KUKA KRL program: EPS_2_25716_MHLP06_A_20250905053030.src

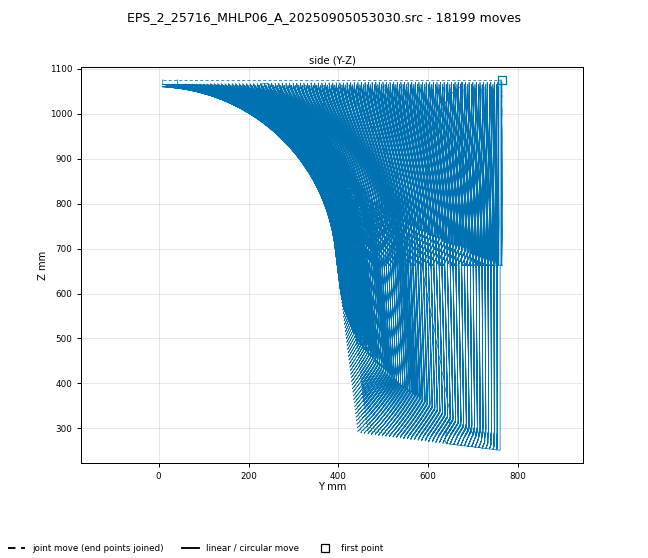
[picture p0: tool path of EPS_2_25716_MHLP06_A_20250905053030.src, 18199 of 18201 moves have a stored position in this frame; points joined in program order, loops and branches not executed]
&ACCESS RVP
&REL 4
&COMMENT QRS 19112012
&PARAM EDITMASK = *
DEF PART()
EXT BAS (BAS_COMMAND :IN,REAL :IN )
INT I
BAS (#INITMOV,0 )

;KUKA QRS Post kuka4.cps  Date:22-06-2017 !

File_ID=2814

QRS_PRE_INIT()

;Init var - Until changes are made in qrs_pre_init
Outlet_Square_prg=0
Inlet_1_Square_prg=0
Inlet_2_Square_prg=0
Inlet_3_Square_prg=0
Inlet_4_Square_prg=0
Inlet_5_Square_prg=0

Outlet_1={X 0.000, Y 514.000, Z 684.500, B 0.000, E1 0.000 }
Inlet_1={X 0.000, Y 514.000, Z 674.500, B 0.000, E1 183.000 }
Outlet_1_type=762
Inlet_1_type=762
;QRS#1=Sidecore dimensions
;QRS#2=750-30" Concrete
;QRS#3=750-30" Concrete
;QRS#4=
;QRS#5=
;QRS#6=
;QRS#7=
;QRS#8=
;QRS#9=S306-42L
;QRS#10=S306-42L
;QRS#11=
;QRS#12=
;QRS#13=
;QRS#14=
;QRS#15=
;QRS#16=1524x152x1524 5'
;QRS#17=EPS Height
;QRS#18=1065,5
;QRS#19=*
;QRS#20= UPDATED VERSION 22-06-2017
;QRS#21=*
Outlet_Square=0550
Inlet_1_Square=0550
Inlet_2_Square=0
Inlet_3_Square=0
Inlet_4_Square=0
Inlet_5_Square=0
Mill_Square=1
Outlet_Square_Prg=266
Inlet_1_Square_prg=266

QRS_INIT()

$ADVANCE=5

; T1
PTP {E1 176.657,E2 176.657}
PTP {X 0,Y 763.394,A -85,B 0,C 180,E1 176.657,E2 176.657,E3 0,E4 0,E5 0,E6 0}
QRS_SPEED_INIT()
LIN {X 0,Y 763.394,Z 1075.5,A -85,B 0,C 180,E1 176.657,E2 176.657,E3 0,E4 0,E5 0,E6 0} C_VEL
LIN {X 0,Y 763.394,Z 665.19,A -85,B 0,C 180,E1 176.657,E2 176.657} C_VEL
LIN {X 0,Y 763.503,Z 663.19,A -85,B 0,C 180,E1 176.807,E2 176.807} C_VEL
LIN {X 0,Y 763.802,Z 663.19,A -85,B 0,C 180,E1 177.187,E2 177.187} C_VEL
LIN {X 0,Y 763.843,Z 663.19,A -85,B 0,C 180,E1 184.692,E2 184.692} C_VEL
LIN {X 0,Y 763.839,Z 663.19,A -85,B 0,C 180,E1 192.28,E2 192.28} C_VEL
LIN {X 0,Y 763.794,Z 663.19,A -85,B 0,C 180,E1 200.096,E2 200.096} C_VEL
LIN {X 0,Y 763.778,Z 663.19,A -85,B 0,C 180,E1 208.327,E2 208.327} C_VEL
LIN {X 0,Y 762.889,Z 663.19,A -85,B 0,C 180,E1 213.338,E2 213.338} C_VEL
LIN {X 0,Y 763.785,Z 663.19,A -85,B 0,C 180,E1 214.937,E2 214.937} C_VEL
LIN {X 0,Y 762.534,Z 663.19,A -85,B 0,C 180,E1 217.329,E2 217.329} C_VEL
LIN {X 0,Y 763.704,Z 663.19,A -85,B 0,C 180,E1 222.138,E2 222.138} C_VEL
LIN {X 0,Y 763.543,Z 663.19,A -85,B 0,C 180,E1 222.564,E2 222.564} C_VEL
LIN {X 0,Y 763.776,Z 663.19,A -85,B 0,C 180,E1 230.266,E2 230.266} C_VEL
LIN {X 0,Y 763.81,Z 663.19,A -85,B 0,C 180,E1 236.912,E2 236.912} C_VEL
LIN {X 0,Y 763.611,Z 663.19,A -85,B 0,C 180,E1 237.107,E2 237.107} C_VEL
LIN {X 0,Y 763.119,Z 663.19,A -85,B 0,C 180,E1 237.178,E2 237.178} C_VEL
LIN {X 0,Y 763.363,Z 714.143,A -85,B 0,C 180,E1 237.755,E2 237.755} C_VEL
LIN {X 0,Y 763.318,Z 729.71,A -85,B 0,C 180,E1 237.961,E2 237.961} C_VEL
LIN {X 0,Y 763.689,Z 748.835,A -85,B 0,C 180,E1 238.314,E2 238.314} C_VEL
LIN {X 0,Y 763.731,Z 766.662,A -85,B 0,C 180,E1 238.702,E2 238.702} C_VEL
LIN {X 0,Y 763.562,Z 784.529,A -85,B 0,C 180,E1 239.155,E2 239.155} C_VEL
LIN {X 0,Y 763.44,Z 791.39,A -85,B 0,C 180,E1 239.353,E2 239.353} C_VEL
LIN {X 0,Y 763.675,Z 803.719,A -85,B 0,C 180,E1 239.742,E2 239.742} C_VEL
LIN {X 0,Y 763.697,Z 820.778,A -85,B 0,C 180,E1 240.333,E2 240.333} C_VEL
LIN {X 0,Y 763.708,Z 837.223,A -85,B 0,C 180,E1 240.974,E2 240.974} C_VEL
LIN {X 0,Y 763.533,Z 854.722,A -85,B 0,C 180,E1 241.73,E2 241.73} C_VEL
LIN {X 0,Y 763.603,Z 871.159,A -85,B 0,C 180,E1 242.528,E2 242.528} C_VEL
LIN {X 0,Y 763.499,Z 886.059,A -85,B 0,C 180,E1 243.314,E2 243.314} C_VEL
LIN {X 0,Y 763.597,Z 901.587,A -85,B 0,C 180,E1 244.22,E2 244.22} C_VEL
LIN {X 0,Y 763.668,Z 915.737,A -85,B 0,C 180,E1 245.118,E2 245.118} C_VEL
LIN {X 0,Y 763.474,Z 930.101,A -85,B 0,C 180,E1 246.101,E2 246.101} C_VEL
LIN {X 0,Y 763.247,Z 942.154,A -85,B 0,C 180,E1 246.988,E2 246.988} C_VEL
LIN {X 0,Y 763.336,Z 956.125,A -85,B 0,C 180,E1 248.123,E2 248.123} C_VEL
LIN {X 0,Y 763.672,Z 967.425,A -85,B 0,C 180,E1 249.12,E2 249.12} C_VEL
LIN {X 0,Y 763.718,Z 974.344,A -85,B 0,C 180,E1 249.772,E2 249.772} C_VEL
LIN {X 0,Y 763.495,Z 980.364,A -85,B 0,C 180,E1 250.349,E2 250.349} C_VEL
LIN {X 0,Y 763.109,Z 990.023,A -85,B 0,C 180,E1 251.332,E2 251.332} C_VEL
LIN {X 0,Y 763.102,Z 1001.366,A -85,B 0,C 180,E1 252.61,E2 252.61} C_VEL
LIN {X 0,Y 763.584,Z 1011.288,A -85,B 0,C 180,E1 253.846,E2 253.846} C_VEL
LIN {X 0,Y 763.803,Z 1015.168,A -85,B 0,C 180,E1 254.372,E2 254.372} C_VEL
LIN {X 0,Y 763.479,Z 1020.327,A -85,B 0,C 180,E1 255.068,E2 255.068} C_VEL
LIN {X 0,Y 762.821,Z 1029.368,A -85,B 0,C 180,E1 256.42,E2 256.42} C_VEL
LIN {X 0,Y 762.79,Z 1036.991,A -85,B 0,C 180,E1 257.703,E2 257.703} C_VEL
LIN {X 0,Y 763.317,Z 1043.373,A -85,B 0,C 180,E1 258.909,E2 258.909} C_VEL
LIN {X 0,Y 763.857,Z 1047.833,A -85,B 0,C 180,E1 259.87,E2 259.87} C_VEL
LIN {X 0,Y 763.425,Z 1050.969,A -85,B 0,C 180,E1 260.578,E2 260.578} C_VEL
LIN {X 0,Y 762.895,Z 1054.781,A -85,B 0,C 180,E1 261.522,E2 261.522} C_VEL
LIN {X 0,Y 762.702,Z 1059.648,A -85,B 0,C 180,E1 262.941,E2 262.941} C_VEL
LIN {X 0,Y 763.282,Z 1063.577,A -85,B 0,C 180,E1 264.362,E2 264.362} C_VEL
LIN {X 0,Y 763.859,Z 1065.587,A -85,B 0,C 180,E1 265.308,E2 265.308} C_VEL
LIN {X 0,Y 763.248,Z 1067.349,A -85,B 0,C 180,E1 266.245,E2 266.245} C_VEL
LIN {X 0,Y 762.721,Z 1068.773,A -85,B 0,C 180,E1 267.183,E2 267.183} C_VEL
LIN {X 0,Y 762.577,Z 1069.998,A -85,B 0,C 180,E1 268.516,E2 268.516} C_VEL
LIN {X 0,Y 762.768,Z 1070.218,A -85,B 0,C 180,E1 269.061,E2 269.061} C_VEL
LIN {X 0,Y 763.872,Z 1070.168,A -85,B 0,C 180,E1 270.937,E2 270.937} C_VEL
LIN {X 0,Y 762.833,Z 1068.771,A -85,B 0,C 180,E1 272.817,E2 272.817} C_VEL
LIN {X 0,Y 762.711,Z 1067.364,A -85,B 0,C 180,E1 273.758,E2 273.758} C_VEL
LIN {X 0,Y 763.16,Z 1064.621,A -85,B 0,C 180,E1 275.167,E2 275.167} C_VEL
LIN {X 0,Y 763.421,Z 1063.574,A -85,B 0,C 180,E1 275.637,E2 275.637} C_VEL
LIN {X 0,Y 763.736,Z 1062.272,A -85,B 0,C 180,E1 276.106,E2 276.106} C_VEL
LIN {X 0,Y 763.75,Z 1060.982,A -85,B 0,C 180,E1 276.577,E2 276.577} C_VEL
LIN {X 0,Y 763.44,Z 1059.643,A -85,B 0,C 180,E1 277.052,E2 277.052} C_VEL
LIN {X 0,Y 762.747,Z 1054.781,A -85,B 0,C 180,E1 278.48,E2 278.48} C_VEL
LIN {X 0,Y 762.808,Z 1048.947,A -85,B 0,C 180,E1 279.905,E2 279.905} C_VEL
LIN {X 0,Y 763.408,Z 1043.373,A -85,B 0,C 180,E1 281.09,E2 281.09} C_VEL
LIN {X 0,Y 763.848,Z 1039.547,A -85,B 0,C 180,E1 281.801,E2 281.801} C_VEL
LIN {X 0,Y 763.464,Z 1035.559,A -85,B 0,C 180,E1 282.541,E2 282.541} C_VEL
LIN {X 0,Y 762.835,Z 1027.394,A -85,B 0,C 180,E1 283.893,E2 283.893} C_VEL
LIN {X 0,Y 762.833,Z 1019.123,A -85,B 0,C 180,E1 285.118,E2 285.118} C_VEL
LIN {X 0,Y 763.436,Z 1009.403,A -85,B 0,C 180,E1 286.402,E2 286.402} C_VEL
LIN {X 0,Y 763.773,Z 1002.371,A -85,B 0,C 180,E1 287.251,E2 287.251} C_VEL
LIN {X 0,Y 763.509,Z 997.07,A -85,B 0,C 180,E1 287.872,E2 287.872} C_VEL
LIN {X 0,Y 763.096,Z 987.878,A -85,B 0,C 180,E1 288.893,E2 288.893} C_VEL
LIN {X 0,Y 762.987,Z 977.021,A -85,B 0,C 180,E1 289.997,E2 289.997} C_VEL
LIN {X 0,Y 763.373,Z 965.026,A -85,B 0,C 180,E1 291.104,E2 291.104} C_VEL
LIN {X 0,Y 763.731,Z 953.245,A -85,B 0,C 180,E1 292.108,E2 292.108} C_VEL
LIN {X 0,Y 763.51,Z 940.467,A -85,B 0,C 180,E1 293.131,E2 293.131} C_VEL
LIN {X 0,Y 763.337,Z 926.48,A -85,B 0,C 180,E1 294.16,E2 294.16} C_VEL
LIN {X 0,Y 763.448,Z 913.778,A -85,B 0,C 180,E1 295.02,E2 295.02} C_VEL
LIN {X 0,Y 763.641,Z 897.91,A -85,B 0,C 180,E1 295.998,E2 295.998} C_VEL
LIN {X 0,Y 763.658,Z 882.443,A -85,B 0,C 180,E1 296.877,E2 296.877} C_VEL
LIN {X 0,Y 763.545,Z 867.236,A -85,B 0,C 180,E1 297.672,E2 297.672} C_VEL
LIN {X 0,Y 763.556,Z 851.419,A -85,B 0,C 180,E1 298.422,E2 298.422} C_VEL
LIN {X 0,Y 763.605,Z 833.293,A -85,B 0,C 180,E1 299.189,E2 299.189} C_VEL
LIN {X 0,Y 763.476,Z 824.344,A -85,B 0,C 180,E1 299.538,E2 299.538} C_VEL
LIN {X 0,Y 763.667,Z 815.688,A -85,B 0,C 180,E1 299.851,E2 299.851} C_VEL
LIN {X 0,Y 763.746,Z 798.997,A -85,B 0,C 180,E1 300.407,E2 300.407} C_VEL
LIN {X 0,Y 763.741,Z 783.59,A -85,B 0,C 180,E1 300.865,E2 300.865} C_VEL
LIN {X 0,Y 763.589,Z 765.456,A -85,B 0,C 180,E1 301.335,E2 301.335} C_VEL
LIN {X 0,Y 763.354,Z 758.258,A -85,B 0,C 180,E1 301.501,E2 301.501} C_VEL
LIN {X 0,Y 763.664,Z 747.28,A -85,B 0,C 180,E1 301.72,E2 301.72} C_VEL
LIN {X 0,Y 763.798,Z 726.383,A -85,B 0,C 180,E1 302.066,E2 302.066} C_VEL
LIN {X 0,Y 763.735,Z 707.916,A -85,B 0,C 180,E1 302.303,E2 302.303} C_VEL
LIN {X 0,Y 763.144,Z 663.19,A -85,B 0,C 180,E1 302.825,E2 302.825} C_VEL
LIN {X 0,Y 763.558,Z 663.19,A -85,B 0,C 180,E1 302.883,E2 302.883} C_VEL
LIN {X 0,Y 763.85,Z 663.19,A -85,B 0,C 180,E1 303.062,E2 303.062} C_VEL
LIN {X 0,Y 763.52,Z 663.19,A -85,B 0,C 180,E1 304.95,E2 304.95} C_VEL
LIN {X 0,Y 763.712,Z 663.19,A -85,B 0,C 180,E1 306.696,E2 306.696} C_VEL
LIN {X 0,Y 763.759,Z 663.19,A -85,B 0,C 180,E1 314.716,E2 314.716} C_VEL
LIN {X 0,Y 763.488,Z 663.19,A -85,B 0,C 180,E1 315.264,E2 315.264} C_VEL
LIN {X 0,Y 763.667,Z 663.19,A -85,B 0,C 180,E1 323.308,E2 323.308} C_VEL
LIN {X 0,Y 762.67,Z 663.19,A -85,B 0,C 180,E1 325.005,E2 325.005} C_VEL
LIN {X 0,Y 762.796,Z 663.19,A -85,B 0,C 180,E1 330.263,E2 330.263} C_VEL
LIN {X 0,Y 763.78,Z 663.19,A -85,B 0,C 180,E1 331.673,E2 331.673} C_VEL
LIN {X 0,Y 763.794,Z 663.19,A -85,B 0,C 180,E1 339.904,E2 339.904} C_VEL
LIN {X 0,Y 763.827,Z 663.19,A -85,B 0,C 180,E1 347.72,E2 347.72} C_VEL
LIN {X 0,Y 763.847,Z 663.19,A -85,B 0,C 180,E1 355.308,E2 355.308} C_VEL
LIN {X 0,Y 763.809,Z 663.19,A -85,B 0,C 180,E1 362.813,E2 362.813} C_VEL
LIN {X 0,Y 763.805,Z 663.19,A -85,B 0,C 180,E1 370.368,E2 370.368} C_VEL
LIN {X 0,Y 763.839,Z 663.19,A -85,B 0,C 180,E1 378.111,E2 378.111} C_VEL
LIN {X 0,Y 762.865,Z 663.19,A -85,B 0,C 180,E1 384.176,E2 384.176} C_VEL
LIN {X 0,Y 763.612,Z 663.19,A -85,B 0,C 180,E1 385.827,E2 385.827} C_VEL
LIN {X 0,Y 763.75,Z 663.19,A -85,B 0,C 180,E1 392.682,E2 392.682} C_VEL
LIN {X 0,Y 763.382,Z 663.19,A -85,B 0,C 180,E1 393.395,E2 393.395} C_VEL
LIN {X 0,Y 763.739,Z 663.19,A -85,B 0,C 180,E1 399.655,E2 399.655} C_VEL
LIN {X 0,Y 763.682,Z 663.19,A -85,B 0,C 180,E1 407.425,E2 407.425} C_VEL
LIN {X 0,Y 763.622,Z 663.19,A -85,B 0,C 180,E1 407.857,E2 407.857} C_VEL
LIN {X 0,Y 763.835,Z 663.19,A -85,B 0,C 180,E1 413.794,E2 413.794} C_VEL
LIN {X 0,Y 763.629,Z 663.19,A -85,B 0,C 180,E1 413.971,E2 413.971} C_VEL
LIN {X 0,Y 761.949,Z 663.19,A -85,B 0,C 180,E1 414.133,E2 414.133} C_VEL
LIN {X 0,Y 762.674,Z 670.746,A -85,B 0,C 180,E1 414.304,E2 414.304} C_VEL
LIN {X 0,Y 763.27,Z 683.05,A -85,B 0,C 180,E1 414.467,E2 414.467} C_VEL
LIN {X 0,Y 763.291,Z 706.143,A -85,B 0,C 180,E1 414.733,E2 414.733} C_VEL
LIN {X 0,Y 763.674,Z 720.884,A -85,B 0,C 180,E1 414.953,E2 414.953} C_VEL
LIN {X 0,Y 763.785,Z 738.788,A -85,B 0,C 180,E1 415.273,E2 415.273} C_VEL
LIN {X 0,Y 763.777,Z 756.953,A -85,B 0,C 180,E1 415.666,E2 415.666} C_VEL
LIN {X 0,Y 763.551,Z 774.753,A -85,B 0,C 180,E1 416.116,E2 416.116} C_VEL
LIN {X 0,Y 763.448,Z 780.911,A -85,B 0,C 180,E1 416.294,E2 416.294} C_VEL
LIN {X 0,Y 763.664,Z 793.266,A -85,B 0,C 180,E1 416.681,E2 416.681} C_VEL
LIN {X 0,Y 763.695,Z 810.232,A -85,B 0,C 180,E1 417.267,E2 417.267} C_VEL
LIN {X 0,Y 763.706,Z 827.815,A -85,B 0,C 180,E1 417.954,E2 417.954} C_VEL
LIN {X 0,Y 763.563,Z 844.112,A -85,B 0,C 180,E1 418.657,E2 418.657} C_VEL
LIN {X 0,Y 763.608,Z 859.823,A -85,B 0,C 180,E1 419.413,E2 419.413} C_VEL
LIN {X 0,Y 763.513,Z 875.27,A -85,B 0,C 180,E1 420.224,E2 420.224} C_VEL
LIN {X 0,Y 763.605,Z 891.803,A -85,B 0,C 180,E1 421.189,E2 421.189} C_VEL
LIN {X 0,Y 763.698,Z 905.659,A -85,B 0,C 180,E1 422.069,E2 422.069} C_VEL
LIN {X 0,Y 763.535,Z 919.141,A -85,B 0,C 180,E1 422.987,E2 422.987} C_VEL
LIN {X 0,Y 763.26,Z 932.57,A -85,B 0,C 180,E1 423.977,E2 423.977} C_VEL
LIN {X 0,Y 763.327,Z 945.733,A -85,B 0,C 180,E1 425.044,E2 425.044} C_VEL
LIN {X 0,Y 763.668,Z 957.774,A -85,B 0,C 180,E1 426.108,E2 426.108} C_VEL
LIN {X 0,Y 763.749,Z 964.577,A -85,B 0,C 180,E1 426.75,E2 426.75} C_VEL
LIN {X 0,Y 763.488,Z 971.081,A -85,B 0,C 180,E1 427.378,E2 427.378} C_VEL
LIN {X 0,Y 763.087,Z 979.912,A -85,B 0,C 180,E1 428.274,E2 428.274} C_VEL
LIN {X 0,Y 762.976,Z 990.113,A -85,B 0,C 180,E1 429.41,E2 429.41} C_VEL
LIN {X 0,Y 763.479,Z 1001.309,A -85,B 0,C 180,E1 430.801,E2 430.801} C_VEL
LIN {X 0,Y 763.844,Z 1007.354,A -85,B 0,C 180,E1 431.62,E2 431.62} C_VEL
LIN {X 0,Y 763.573,Z 1011.028,A -85,B 0,C 180,E1 432.129,E2 432.129} C_VEL
LIN {X 0,Y 762.949,Z 1019.161,A -85,B 0,C 180,E1 433.343,E2 433.343} C_VEL
LIN {X 0,Y 762.76,Z 1025.695,A -85,B 0,C 180,E1 434.425,E2 434.425} C_VEL
LIN {X 0,Y 763.186,Z 1032.951,A -85,B 0,C 180,E1 435.781,E2 435.781} C_VEL
LIN {X 0,Y 763.744,Z 1037.559,A -85,B 0,C 180,E1 436.765,E2 436.765} C_VEL
LIN {X 0,Y 763.737,Z 1039.417,A -85,B 0,C 180,E1 437.162,E2 437.162} C_VEL
LIN {X 0,Y 762.866,Z 1045.491,A -85,B 0,C 180,E1 438.663,E2 438.663} C_VEL
LIN {X 0,Y 762.68,Z 1050.25,A -85,B 0,C 180,E1 440.093,E2 440.093} C_VEL
LIN {X 0,Y 763.274,Z 1054.066,A -85,B 0,C 180,E1 441.526,E2 441.526} C_VEL
LIN {X 0,Y 763.845,Z 1056.046,A -85,B 0,C 180,E1 442.479,E2 442.479} C_VEL
LIN {X 0,Y 763.25,Z 1057.677,A -85,B 0,C 180,E1 443.419,E2 443.419} C_VEL
LIN {X 0,Y 762.729,Z 1059.001,A -85,B 0,C 180,E1 444.358,E2 444.358} C_VEL
LIN {X 0,Y 762.57,Z 1059.845,A -85,B 0,C 180,E1 445.3,E2 445.3} C_VEL
LIN {X 0,Y 762.768,Z 1060.283,A -85,B 0,C 180,E1 446.236,E2 446.236} C_VEL
LIN {X 0,Y 763.261,Z 1060.412,A -85,B 0,C 180,E1 447.185,E2 447.185} C_VEL
LIN {X 0,Y 763.773,Z 1060.049,A -85,B 0,C 180,E1 448.312,E2 448.312} C_VEL
LIN {X 0,Y 762.916,Z 1058.708,A -85,B 0,C 180,E1 449.812,E2 449.812} C_VEL
LIN {X 0,Y 762.704,Z 1057.026,A -85,B 0,C 180,E1 450.939,E2 450.939} C_VEL
LIN {X 0,Y 763.033,Z 1054.747,A -85,B 0,C 180,E1 452.065,E2 452.065} C_VEL
LIN {X 0,Y 763.434,Z 1052.961,A -85,B 0,C 180,E1 452.815,E2 452.815} C_VEL
LIN {X 0,Y 763.825,Z 1050.803,A -85,B 0,C 180,E1 453.596,E2 453.596} C_VEL
LIN {X 0,Y 763.187,Z 1047.332,A -85,B 0,C 180,E1 454.696,E2 454.696} C_VEL
LIN {X 0,Y 762.935,Z 1045.751,A -85,B 0,C 180,E1 455.169,E2 455.169} C_VEL
LIN {X 0,Y 762.766,Z 1039.129,A -85,B 0,C 180,E1 456.822,E2 456.822} C_VEL
LIN {X 0,Y 763.285,Z 1033.601,A -85,B 0,C 180,E1 458,E2 458} C_VEL
LIN {X 0,Y 763.86,Z 1028.555,A -85,B 0,C 180,E1 458.941,E2 458.941} C_VEL
LIN {X 0,Y 763.483,Z 1024.574,A -85,B 0,C 180,E1 459.659,E2 459.659} C_VEL
LIN {X 0,Y 762.931,Z 1017.317,A -85,B 0,C 180,E1 460.858,E2 460.858} C_VEL
LIN {X 0,Y 762.854,Z 1009.247,A -85,B 0,C 180,E1 462.056,E2 462.056} C_VEL
LIN {X 0,Y 763.43,Z 998.964,A -85,B 0,C 180,E1 463.41,E2 463.41} C_VEL
LIN {X 0,Y 763.814,Z 992.361,A -85,B 0,C 180,E1 464.207,E2 464.207} C_VEL
LIN {X 0,Y 763.552,Z 986.364,A -85,B 0,C 180,E1 464.905,E2 464.905} C_VEL
LIN {X 0,Y 763.202,Z 978.727,A -85,B 0,C 180,E1 465.759,E2 465.759} C_VEL
LIN {X 0,Y 763.026,Z 967.557,A -85,B 0,C 180,E1 466.901,E2 466.901} C_VEL
LIN {X 0,Y 763.363,Z 955.721,A -85,B 0,C 180,E1 467.999,E2 467.999} C_VEL
LIN {X 0,Y 763.745,Z 942.465,A -85,B 0,C 180,E1 469.125,E2 469.125} C_VEL
LIN {X 0,Y 763.517,Z 930.218,A -85,B 0,C 180,E1 470.104,E2 470.104} C_VEL
LIN {X 0,Y 763.287,Z 916.729,A -85,B 0,C 180,E1 471.1,E2 471.1} C_VEL
LIN {X 0,Y 763.377,Z 902.542,A -85,B 0,C 180,E1 472.055,E2 472.055} C_VEL
LIN {X 0,Y 763.626,Z 888.226,A -85,B 0,C 180,E1 472.936,E2 472.936} C_VEL
LIN {X 0,Y 763.684,Z 872.5,A -85,B 0,C 180,E1 473.828,E2 473.828} C_VEL
LIN {X 0,Y 763.623,Z 856.934,A -85,B 0,C 180,E1 474.639,E2 474.639} C_VEL
LIN {X 0,Y 763.629,Z 840.802,A -85,B 0,C 180,E1 475.4,E2 475.4} C_VEL
LIN {X 0,Y 763.624,Z 823.946,A -85,B 0,C 180,E1 476.118,E2 476.118} C_VEL
LIN {X 0,Y 763.519,Z 814.426,A -85,B 0,C 180,E1 476.489,E2 476.489} C_VEL
LIN {X 0,Y 763.706,Z 805.542,A -85,B 0,C 180,E1 476.809,E2 476.809} C_VEL
LIN {X 0,Y 763.748,Z 788.836,A -85,B 0,C 180,E1 477.367,E2 477.367} C_VEL
LIN {X 0,Y 763.74,Z 771.331,A -85,B 0,C 180,E1 477.88,E2 477.88} C_VEL
LIN {X 0,Y 763.608,Z 752.724,A -85,B 0,C 180,E1 478.35,E2 478.35} C_VEL
LIN {X 0,Y 763.364,Z 742.185,A -85,B 0,C 180,E1 478.585,E2 478.585} C_VEL
LIN {X 0,Y 763.599,Z 733.423,A -85,B 0,C 180,E1 478.746,E2 478.746} C_VEL
LIN {X 0,Y 763.746,Z 718.002,A -85,B 0,C 180,E1 479.002,E2 479.002} C_VEL
LIN {X 0,Y 763.66,Z 695.951,A -85,B 0,C 180,E1 479.283,E2 479.283} C_VEL
LIN {X 0,Y 763.248,Z 663.19,A -85,B 0,C 180,E1 479.663,E2 479.663} C_VEL
LIN {X 0,Y 763.483,Z 663.19,A -85,B 0,C 180,E1 479.696,E2 479.696} C_VEL
LIN {X 0,Y 763.798,Z 663.19,A -85,B 0,C 180,E1 479.868,E2 479.868} C_VEL
LIN {X 0,Y 762.898,Z 663.19,A -85,B 0,C 180,E1 484.983,E2 484.983} C_VEL
LIN {X 0,Y 763.644,Z 663.19,A -85,B 0,C 180,E1 486.689,E2 486.689} C_VEL
LIN {X 0,Y 763.687,Z 663.19,A -85,B 0,C 180,E1 494.721,E2 494.721} C_VEL
LIN {X 0,Y 763.478,Z 663.19,A -85,B 0,C 180,E1 495.263,E2 495.263} C_VEL
LIN {X 0,Y 762.367,Z 663.19,A -85,B 0,C 180,E1 500.394,E2 500.394} C_VEL
LIN {X 0,Y 763.72,Z 663.19,A -85,B 0,C 180,E1 502.739,E2 502.739} C_VEL
LIN {X 0,Y 763.638,Z 663.19,A -85,B 0,C 180,E1 510.152,E2 510.152} C_VEL
LIN {X 0,Y 762.933,Z 663.19,A -85,B 0,C 180,E1 511.639,E2 511.639} C_VEL
LIN {X 0,Y 763.821,Z 663.19,A -85,B 0,C 180,E1 517.895,E2 517.895} C_VEL
LIN {X 0,Y 763.451,Z 663.19,A -85,B 0,C 180,E1 524.967,E2 524.967} C_VEL
LIN {X 0,Y 763.654,Z 663.19,A -85,B 0,C 180,E1 525.79,E2 525.79} C_VEL
LIN {X 0,Y 763.811,Z 663.19,A -85,B 0,C 180,E1 529.632,E2 529.632} C_VEL
LIN {X 0,Y 763.503,Z 663.19,A -85,B 0,C 180,E1 536.807,E2 536.807} C_VEL
LIN {X 0,Y 754.48,Z 663.19,A -85,B 0,C 180,E1 539.404,E2 539.404} C_VEL
LIN {X 0,Y 754.687,Z 663.19,A -85,B 0,C 180,E1 546.363,E2 546.363} C_VEL
LIN {X 0,Y 754.972,Z 663.19,A -85,B 0,C 180,E1 553.38,E2 553.38} C_VEL
LIN {X 0,Y 755.058,Z 663.19,A -85,B 0,C 180,E1 560.953,E2 560.953} C_VEL
LIN {X 0,Y 755.058,Z 663.19,A -85,B 0,C 180,E1 569.519,E2 569.519} C_VEL
LIN {X 0,Y 754.873,Z 663.19,A -85,B 0,C 180,E1 576.396,E2 576.396} C_VEL
LIN {X 0,Y 755.272,Z 663.19,A -85,B 0,C 180,E1 582.876,E2 582.876} C_VEL
LIN {X 0,Y 755.409,Z 663.19,A -85,B 0,C 180,E1 590.778,E2 590.778} C_VEL
LIN {X 0,Y 755.916,Z 664.759,A -85,B 0,C 180,E1 596.843,E2 596.843} C_VEL
LIN {X 0,Y 756.868,Z 759.718,A -85,B 0,C 180,E1 598.229,E2 598.229} C_VEL
LIN {X 0,Y 756.569,Z 829.969,A -85,B 0,C 180,E1 600.384,E2 600.384} C_VEL
LIN {X 0,Y 756.114,Z 898.18,A -85,B 0,C 180,E1 603.739,E2 603.739} C_VEL
LIN {X 0,Y 755.607,Z 957.987,A -85,B 0,C 180,E1 608.051,E2 608.051} C_VEL
LIN {X 0,Y 755.379,Z 1006.638,A -85,B 0,C 180,E1 613.077,E2 613.077} C_VEL
LIN {X 0,Y 755.094,Z 1041.42,A -85,B 0,C 180,E1 618.415,E2 618.415} C_VEL
LIN {X 0,Y 754.949,Z 1061.847,A -85,B 0,C 180,E1 623.658,E2 623.658} C_VEL
LIN {X 0,Y 754.595,Z 1069.802,A -85,B 0,C 180,E1 628.273,E2 628.273} C_VEL
LIN {X 0,Y 754.847,Z 1068.731,A -85,B 0,C 180,E1 632.879,E2 632.879} C_VEL
LIN {X 0,Y 755.199,Z 1058.413,A -85,B 0,C 180,E1 637.5,E2 637.5} C_VEL
LIN {X 0,Y 755.225,Z 1033.216,A -85,B 0,C 180,E1 643.073,E2 643.073} C_VEL
LIN {X 0,Y 755.422,Z 993.868,A -85,B 0,C 180,E1 648.431,E2 648.431} C_VEL
LIN {X 0,Y 755.875,Z 942.929,A -85,B 0,C 180,E1 653.186,E2 653.186} C_VEL
LIN {X 0,Y 756.271,Z 881.314,A -85,B 0,C 180,E1 657.221,E2 657.221} C_VEL
LIN {X 0,Y 756.618,Z 813.428,A -85,B 0,C 180,E1 660.236,E2 660.236} C_VEL
LIN {X 0,Y 756.926,Z 740.759,A -85,B 0,C 180,E1 662.151,E2 662.151} C_VEL
LIN {X 0,Y 755.817,Z 663.19,A -85,B 0,C 180,E1 663.186,E2 663.186} C_VEL
LIN {X 0,Y 754.086,Z 663.19,A -85,B 0,C 180,E1 669.305,E2 669.305} C_VEL
LIN {X 0,Y 754.833,Z 663.19,A -85,B 0,C 180,E1 676.058,E2 676.058} C_VEL
LIN {X 0,Y 754.921,Z 663.19,A -85,B 0,C 180,E1 684.442,E2 684.442} C_VEL
LIN {X 0,Y 755.641,Z 663.19,A -85,B 0,C 180,E1 691.82,E2 691.82} C_VEL
LIN {X 0,Y 755.202,Z 663.19,A -85,B 0,C 180,E1 700.62,E2 700.62} C_VEL
LIN {X 0,Y 754.916,Z 663.19,A -85,B 0,C 180,E1 708.976,E2 708.976} C_VEL
LIN {X 0,Y 755.342,Z 663.19,A -85,B 0,C 180,E1 715.955,E2 715.955} C_VEL
LIN {X 0,Y 754.915,Z 663.19,A -85,B 0,C 180,E1 724.023,E2 724.023} C_VEL
LIN {X 0,Y 755.309,Z 663.19,A -85,B 0,C 180,E1 730.993,E2 730.993} C_VEL
LIN {X 0,Y 754.961,Z 663.19,A -85,B 0,C 180,E1 739.36,E2 739.36} C_VEL
LIN {X 0,Y 754.93,Z 663.19,A -85,B 0,C 180,E1 746.881,E2 746.881} C_VEL
LIN {X 0,Y 755.271,Z 663.19,A -85,B 0,C 180,E1 753.568,E2 753.568} C_VEL
LIN {X 0,Y 754.686,Z 663.19,A -85,B 0,C 180,E1 761.105,E2 761.105} C_VEL
LIN {X 0,Y 755.062,Z 663.19,A -85,B 0,C 180,E1 768.902,E2 768.902} C_VEL
LIN {X 0,Y 754.972,Z 663.19,A -85,B 0,C 180,E1 773.838,E2 773.838} C_VEL
LIN {X 0,Y 756.929,Z 755.494,A -85,B 0,C 180,E1 775.313,E2 775.313} C_VEL
LIN {X 0,Y 756.585,Z 826.044,A -85,B 0,C 180,E1 777.578,E2 777.578} C_VEL
LIN {X 0,Y 756.13,Z 892.372,A -85,B 0,C 180,E1 780.952,E2 780.952} C_VEL
LIN {X 0,Y 755.702,Z 952.369,A -85,B 0,C 180,E1 785.394,E2 785.394} C_VEL
LIN {X 0,Y 755.483,Z 1000.435,A -85,B 0,C 180,E1 790.506,E2 790.506} C_VEL
LIN {X 0,Y 755.342,Z 1034.832,A -85,B 0,C 180,E1 796.059,E2 796.059} C_VEL
LIN {X 0,Y 755.482,Z 1055.025,A -85,B 0,C 180,E1 801.923,E2 801.923} C_VEL
LIN {X 0,Y 755.24,Z 1060.458,A -85,B 0,C 180,E1 807.122,E2 807.122} C_VEL
LIN {X 0,Y 755.477,Z 1052.976,A -85,B 0,C 180,E1 812.876,E2 812.876} C_VEL
LIN {X 0,Y 755.692,Z 1030.759,A -85,B 0,C 180,E1 818.656,E2 818.656} C_VEL
LIN {X 0,Y 755.905,Z 993.718,A -85,B 0,C 180,E1 824.226,E2 824.226} C_VEL
LIN {X 0,Y 756.037,Z 944.765,A -85,B 0,C 180,E1 829.174,E2 829.174} C_VEL
LIN {X 0,Y 756.205,Z 884.806,A -85,B 0,C 180,E1 833.409,E2 833.409} C_VEL
LIN {X 0,Y 756.415,Z 815.296,A -85,B 0,C 180,E1 836.76,E2 836.76} C_VEL
LIN {X 0,Y 756.577,Z 740.886,A -85,B 0,C 180,E1 838.93,E2 838.93} C_VEL
LIN {X 0,Y 755.622,Z 663.19,A -85,B 0,C 180,E1 840.119,E2 840.119} C_VEL
LIN {X 0,Y 754.751,Z 663.19,A -85,B 0,C 180,E1 847.791,E2 847.791} C_VEL
LIN {X 0,Y 754.876,Z 663.19,A -85,B 0,C 180,E1 856.096,E2 856.096} C_VEL
LIN {X 0,Y 755.027,Z 663.19,A -85,B 0,C 180,E1 863.644,E2 863.644} C_VEL
LIN {X 0,Y 754.844,Z 663.19,A -85,B 0,C 180,E1 871.816,E2 871.816} C_VEL
LIN {X 0,Y 754.774,Z 663.19,A -85,B 0,C 180,E1 879.409,E2 879.409} C_VEL
LIN {X 0,Y 755.383,Z 663.19,A -85,B 0,C 180,E1 886.811,E2 886.811} C_VEL
LIN {X 0,Y 754.166,Z 663.19,A -85,B 0,C 180,E1 893.658,E2 893.658} C_VEL
LIN {X 0,Y 755.008,Z 663.19,A -85,B 0,C 180,E1 898.285,E2 898.285} C_VEL
LIN {X 0,Y 754.48,Z 663.19,A -85,B 0,C 180,E1 899.404,E2 899.404} C_VEL
LIN {X 0,Y 746.358,Z 663.19,A -85,B 0,C 180,E1 902.034,E2 902.034} C_VEL
LIN {X 0,Y 746.257,Z 663.19,A -85,B 0,C 180,E1 907.61,E2 907.61} C_VEL
LIN {X 0,Y 746.872,Z 663.19,A -85,B 0,C 180,E1 913.528,E2 913.528} C_VEL
LIN {X 0,Y 747.144,Z 663.19,A -85,B 0,C 180,E1 920.838,E2 920.838} C_VEL
LIN {X 0,Y 747.49,Z 663.19,A -85,B 0,C 180,E1 928.515,E2 928.515} C_VEL
LIN {X 0,Y 747.446,Z 663.19,A -85,B 0,C 180,E1 935.377,E2 935.377} C_VEL
LIN {X 0,Y 747.243,Z 663.19,A -85,B 0,C 180,E1 942.896,E2 942.896} C_VEL
LIN {X 0,Y 746.902,Z 663.19,A -85,B 0,C 180,E1 951.74,E2 951.74} C_VEL
LIN {X 0,Y 747.708,Z 665.181,A -85,B 0,C 180,E1 956.436,E2 956.436} C_VEL
LIN {X 0,Y 749.825,Z 699.861,A -85,B 0,C 180,E1 956.932,E2 956.932} C_VEL
LIN {X 0,Y 749.856,Z 774.935,A -85,B 0,C 180,E1 958.271,E2 958.271} C_VEL
LIN {X 0,Y 749.273,Z 845.914,A -85,B 0,C 180,E1 960.743,E2 960.743} C_VEL
LIN {X 0,Y 748.603,Z 911.358,A -85,B 0,C 180,E1 964.293,E2 964.293} C_VEL
LIN {X 0,Y 748.101,Z 969.045,A -85,B 0,C 180,E1 968.82,E2 968.82} C_VEL
LIN {X 0,Y 747.915,Z 1015.785,A -85,B 0,C 180,E1 974.115,E2 974.115} C_VEL
LIN {X 0,Y 747.661,Z 1047.079,A -85,B 0,C 180,E1 979.483,E2 979.483} C_VEL
LIN {X 0,Y 747.775,Z 1065.919,A -85,B 0,C 180,E1 985.348,E2 985.348} C_VEL
LIN {X 0,Y 747.602,Z 1070.338,A -85,B 0,C 180,E1 990.581,E2 990.581} C_VEL
LIN {X 0,Y 747.718,Z 1061.845,A -85,B 0,C 180,E1 996.405,E2 996.405} C_VEL
LIN {X 0,Y 747.658,Z 1038.316,A -85,B 0,C 180,E1 1002.296,E2 1002.296} C_VEL
LIN {X 0,Y 747.847,Z 1001.03,A -85,B 0,C 180,E1 1007.799,E2 1007.799} C_VEL
LIN {X 0,Y 748.229,Z 950.883,A -85,B 0,C 180,E1 1012.784,E2 1012.784} C_VEL
LIN {X 0,Y 748.843,Z 890.489,A -85,B 0,C 180,E1 1016.99,E2 1016.99} C_VEL
LIN {X 0,Y 749.401,Z 822.492,A -85,B 0,C 180,E1 1020.224,E2 1020.224} C_VEL
LIN {X 0,Y 749.952,Z 749.891,A -85,B 0,C 180,E1 1022.313,E2 1022.313} C_VEL
LIN {X 0,Y 748.098,Z 665.576,A -85,B 0,C 180,E1 1023.54,E2 1023.54} C_VEL
LIN {X 0,Y 747.646,Z 663.19,A -85,B 0,C 180,E1 1023.902,E2 1023.902} C_VEL
LIN {X 0,Y 746.095,Z 663.19,A -85,B 0,C 180,E1 1032.034,E2 1032.034} C_VEL
LIN {X 0,Y 746.774,Z 663.19,A -85,B 0,C 180,E1 1036.127,E2 1036.127} C_VEL
LIN {X 0,Y 746.86,Z 663.19,A -85,B 0,C 180,E1 1044.591,E2 1044.591} C_VEL
LIN {X 0,Y 746.864,Z 663.19,A -85,B 0,C 180,E1 1052.776,E2 1052.776} C_VEL
LIN {X 0,Y 747.163,Z 663.19,A -85,B 0,C 180,E1 1060.691,E2 1060.691} C_VEL
LIN {X 0,Y 746.994,Z 663.19,A -85,B 0,C 180,E1 1068.858,E2 1068.858} C_VEL
LIN {X 0,Y 747.357,Z 663.19,A -85,B 0,C 180,E1 1075.911,E2 1075.911} C_VEL
LIN {X 0,Y 746.882,Z 663.19,A -85,B 0,C 180,E1 1084.066,E2 1084.066} C_VEL
LIN {X 0,Y 747.221,Z 663.19,A -85,B 0,C 180,E1 1091.113,E2 1091.113} C_VEL
LIN {X 0,Y 746.849,Z 663.19,A -85,B 0,C 180,E1 1099.579,E2 1099.579} C_VEL
LIN {X 0,Y 746.772,Z 663.19,A -85,B 0,C 180,E1 1107.199,E2 1107.199} C_VEL
LIN {X 0,Y 746.743,Z 663.19,A -85,B 0,C 180,E1 1114.67,E2 1114.67} C_VEL
LIN {X 0,Y 746.554,Z 663.19,A -85,B 0,C 180,E1 1121.34,E2 1121.34} C_VEL
LIN {X 0,Y 747.129,Z 663.19,A -85,B 0,C 180,E1 1128.727,E2 1128.727} C_VEL
LIN {X 0,Y 747.748,Z 664.557,A -85,B 0,C 180,E1 1133.498,E2 1133.498} C_VEL
LIN {X 0,Y 750.031,Z 757.212,A -85,B 0,C 180,E1 1135.033,E2 1135.033} C_VEL
LIN {X 0,Y 749.44,Z 826.899,A -85,B 0,C 180,E1 1137.308,E2 1137.308} C_VEL
LIN {X 0,Y 748.676,Z 893.608,A -85,B 0,C 180,E1 1140.753,E2 1140.753} C_VEL
LIN {X 0,Y 747.955,Z 953.013,A -85,B 0,C 180,E1 1145.216,E2 1145.216} C_VEL
LIN {X 0,Y 747.532,Z 1000.165,A -85,B 0,C 180,E1 1150.29,E2 1150.29} C_VEL
LIN {X 0,Y 747.315,Z 1034.676,A -85,B 0,C 180,E1 1155.907,E2 1155.907} C_VEL
LIN {X 0,Y 747.453,Z 1054.956,A -85,B 0,C 180,E1 1161.835,E2 1161.835} C_VEL
LIN {X 0,Y 747.215,Z 1060.468,A -85,B 0,C 180,E1 1167.092,E2 1167.092} C_VEL
LIN {X 0,Y 747.505,Z 1053.064,A -85,B 0,C 180,E1 1172.907,E2 1172.907} C_VEL
LIN {X 0,Y 747.757,Z 1030.935,A -85,B 0,C 180,E1 1178.748,E2 1178.748} C_VEL
LIN {X 0,Y 748.004,Z 993.998,A -85,B 0,C 180,E1 1184.379,E2 1184.379} C_VEL
LIN {X 0,Y 748.314,Z 945.84,A -85,B 0,C 180,E1 1189.32,E2 1189.32} C_VEL
LIN {X 0,Y 748.795,Z 886.394,A -85,B 0,C 180,E1 1193.598,E2 1193.598} C_VEL
LIN {X 0,Y 749.292,Z 817.869,A -85,B 0,C 180,E1 1196.971,E2 1196.971} C_VEL
LIN {X 0,Y 749.684,Z 743.698,A -85,B 0,C 180,E1 1199.198,E2 1199.198} C_VEL
LIN {X 0,Y 748.299,Z 666.762,A -85,B 0,C 180,E1 1200.359,E2 1200.359} C_VEL
LIN {X 0,Y 747.354,Z 663.19,A -85,B 0,C 180,E1 1200.536,E2 1200.536} C_VEL
LIN {X 0,Y 746.341,Z 663.19,A -85,B 0,C 180,E1 1208.489,E2 1208.489} C_VEL
LIN {X 0,Y 746.854,Z 663.19,A -85,B 0,C 180,E1 1216.119,E2 1216.119} C_VEL
LIN {X 0,Y 747.147,Z 663.19,A -85,B 0,C 180,E1 1223.292,E2 1223.292} C_VEL
LIN {X 0,Y 746.733,Z 663.19,A -85,B 0,C 180,E1 1232.051,E2 1232.051} C_VEL
LIN {X 0,Y 746.917,Z 663.19,A -85,B 0,C 180,E1 1239.183,E2 1239.183} C_VEL
LIN {X 0,Y 747.334,Z 663.19,A -85,B 0,C 180,E1 1247.7,E2 1247.7} C_VEL
LIN {X 0,Y 747.724,Z 663.19,A -85,B 0,C 180,E1 1257.104,E2 1257.104} C_VEL
LIN {X 0,Y 746.358,Z 663.19,A -85,B 0,C 180,E1 1262.034,E2 1262.034} C_VEL
LIN {X 0,Y 739.292,Z 663.19,A -85,B 0,C 180,E1 1264.716,E2 1264.716} C_VEL
LIN {X 0,Y 738.776,Z 663.19,A -85,B 0,C 180,E1 1273.679,E2 1273.679} C_VEL
LIN {X 0,Y 738.951,Z 663.19,A -85,B 0,C 180,E1 1281.08,E2 1281.08} C_VEL
LIN {X 0,Y 739.107,Z 663.19,A -85,B 0,C 180,E1 1289.313,E2 1289.313} C_VEL
LIN {X 0,Y 739.158,Z 663.19,A -85,B 0,C 180,E1 1295.87,E2 1295.87} C_VEL
LIN {X 0,Y 738.836,Z 663.19,A -85,B 0,C 180,E1 1303.504,E2 1303.504} C_VEL
LIN {X 0,Y 739.061,Z 663.19,A -85,B 0,C 180,E1 1311.259,E2 1311.259} C_VEL
LIN {X 0,Y 739.37,Z 664.769,A -85,B 0,C 180,E1 1316.001,E2 1316.001} C_VEL
LIN {X 0,Y 743.086,Z 678.117,A -85,B 0,C 180,E1 1316.346,E2 1316.346} C_VEL
LIN {X 0,Y 743.192,Z 762.398,A -85,B 0,C 180,E1 1317.632,E2 1317.632} C_VEL
LIN {X 0,Y 742.349,Z 832.082,A -85,B 0,C 180,E1 1319.842,E2 1319.842} C_VEL
LIN {X 0,Y 741.245,Z 900.309,A -85,B 0,C 180,E1 1323.301,E2 1323.301} C_VEL
LIN {X 0,Y 740.163,Z 959.751,A -85,B 0,C 180,E1 1327.727,E2 1327.727} C_VEL
LIN {X 0,Y 739.569,Z 1007.861,A -85,B 0,C 180,E1 1332.858,E2 1332.858} C_VEL
LIN {X 0,Y 739.213,Z 1042.968,A -85,B 0,C 180,E1 1338.463,E2 1338.463} C_VEL
LIN {X 0,Y 739.175,Z 1063.415,A -85,B 0,C 180,E1 1344.113,E2 1344.113} C_VEL
LIN {X 0,Y 738.928,Z 1070.338,A -85,B 0,C 180,E1 1349.412,E2 1349.412} C_VEL
LIN {X 0,Y 739.097,Z 1065.331,A -85,B 0,C 180,E1 1354.995,E2 1354.995} C_VEL
LIN {X 0,Y 739.191,Z 1047.075,A -85,B 0,C 180,E1 1360.64,E2 1360.64} C_VEL
LIN {X 0,Y 739.499,Z 1014.681,A -85,B 0,C 180,E1 1366.224,E2 1366.224} C_VEL
LIN {X 0,Y 740.175,Z 968.384,A -85,B 0,C 180,E1 1371.482,E2 1371.482} C_VEL
LIN {X 0,Y 741.068,Z 910.926,A -85,B 0,C 180,E1 1376.016,E2 1376.016} C_VEL
LIN {X 0,Y 742.052,Z 843.203,A -85,B 0,C 180,E1 1379.691,E2 1379.691} C_VEL
LIN {X 0,Y 742.92,Z 770.56,A -85,B 0,C 180,E1 1382.176,E2 1382.176} C_VEL
LIN {X 0,Y 743.285,Z 689.976,A -85,B 0,C 180,E1 1383.509,E2 1383.509} C_VEL
LIN {X 0,Y 741.024,Z 667.635,A -85,B 0,C 180,E1 1383.88,E2 1383.88} C_VEL
LIN {X 0,Y 739.631,Z 663.19,A -85,B 0,C 180,E1 1384.071,E2 1384.071} C_VEL
LIN {X 0,Y 738.78,Z 663.19,A -85,B 0,C 180,E1 1393.442,E2 1393.442} C_VEL
LIN {X 0,Y 738.884,Z 663.19,A -85,B 0,C 180,E1 1402.685,E2 1402.685} C_VEL
LIN {X 0,Y 739.077,Z 663.19,A -85,B 0,C 180,E1 1412.465,E2 1412.465} C_VEL
LIN {X 0,Y 738.715,Z 663.19,A -85,B 0,C 180,E1 1421.416,E2 1421.416} C_VEL
LIN {X 0,Y 739.042,Z 663.19,A -85,B 0,C 180,E1 1428.736,E2 1428.736} C_VEL
LIN {X 0,Y 739.353,Z 663.19,A -85,B 0,C 180,E1 1435.867,E2 1435.867} C_VEL
LIN {X 0,Y 738.851,Z 663.19,A -85,B 0,C 180,E1 1444.11,E2 1444.11} C_VEL
LIN {X 0,Y 739.122,Z 663.19,A -85,B 0,C 180,E1 1451.237,E2 1451.237} C_VEL
LIN {X 0,Y 739.471,Z 663.19,A -85,B 0,C 180,E1 1458.537,E2 1458.537} C_VEL
LIN {X 0,Y 738.903,Z 663.19,A -85,B 0,C 180,E1 1466.781,E2 1466.781} C_VEL
LIN {X 0,Y 738.856,Z 663.19,A -85,B 0,C 180,E1 1474.381,E2 1474.381} C_VEL
LIN {X 0,Y 738.499,Z 663.19,A -85,B 0,C 180,E1 1481.454,E2 1481.454} C_VEL
LIN {X 0,Y 739.216,Z 663.19,A -85,B 0,C 180,E1 1488.522,E2 1488.522} C_VEL
LIN {X 0,Y 739.471,Z 664.534,A -85,B 0,C 180,E1 1493.073,E2 1493.073} C_VEL
LIN {X 0,Y 743.128,Z 687.641,A -85,B 0,C 180,E1 1493.525,E2 1493.525} C_VEL
LIN {X 0,Y 742.99,Z 765.98,A -85,B 0,C 180,E1 1494.925,E2 1494.925} C_VEL
LIN {X 0,Y 742.058,Z 838.032,A -85,B 0,C 180,E1 1497.48,E2 1497.48} C_VEL
LIN {X 0,Y 741.157,Z 904.279,A -85,B 0,C 180,E1 1501.161,E2 1501.161} C_VEL
LIN {X 0,Y 740.34,Z 961.633,A -85,B 0,C 180,E1 1505.795,E2 1505.795} C_VEL
LIN {X 0,Y 739.868,Z 1006.718,A -85,B 0,C 180,E1 1511.022,E2 1511.022} C_VEL
LIN {X 0,Y 739.756,Z 1038.938,A -85,B 0,C 180,E1 1516.735,E2 1516.735} C_VEL
LIN {X 0,Y 739.717,Z 1056.105,A -85,B 0,C 180,E1 1522.342,E2 1522.342} C_VEL
LIN {X 0,Y 739.71,Z 1060.138,A -85,B 0,C 180,E1 1528.238,E2 1528.238} C_VEL
LIN {X 0,Y 739.533,Z 1050.029,A -85,B 0,C 180,E1 1534.115,E2 1534.115} C_VEL
LIN {X 0,Y 739.457,Z 1024.813,A -85,B 0,C 180,E1 1540.038,E2 1540.038} C_VEL
LIN {X 0,Y 739.764,Z 985.685,A -85,B 0,C 180,E1 1545.582,E2 1545.582} C_VEL
LIN {X 0,Y 740.556,Z 934.394,A -85,B 0,C 180,E1 1550.528,E2 1550.528} C_VEL
LIN {X 0,Y 741.62,Z 872.177,A -85,B 0,C 180,E1 1554.713,E2 1554.713} C_VEL
LIN {X 0,Y 742.618,Z 803.996,A -85,B 0,C 180,E1 1557.803,E2 1557.803} C_VEL
LIN {X 0,Y 743.233,Z 731.679,A -85,B 0,C 180,E1 1559.756,E2 1559.756} C_VEL
LIN {X 0,Y 741.324,Z 668.547,A -85,B 0,C 180,E1 1560.695,E2 1560.695} C_VEL
LIN {X 0,Y 739.137,Z 663.19,A -85,B 0,C 180,E1 1560.978,E2 1560.978} C_VEL
LIN {X 0,Y 738.698,Z 663.19,A -85,B 0,C 180,E1 1567.737,E2 1567.737} C_VEL
LIN {X 0,Y 738.637,Z 663.19,A -85,B 0,C 180,E1 1576.516,E2 1576.516} C_VEL
LIN {X 0,Y 738.711,Z 663.19,A -85,B 0,C 180,E1 1584.178,E2 1584.178} C_VEL
LIN {X 0,Y 738.993,Z 663.19,A -85,B 0,C 180,E1 1591.156,E2 1591.156} C_VEL
LIN {X 0,Y 738.979,Z 663.19,A -85,B 0,C 180,E1 1599.015,E2 1599.015} C_VEL
LIN {X 0,Y 739.326,Z 663.19,A -85,B 0,C 180,E1 1607.565,E2 1607.565} C_VEL
LIN {X 0,Y 739.685,Z 663.19,A -85,B 0,C 180,E1 1617.072,E2 1617.072} C_VEL
LIN {X 0,Y 739.292,Z 663.19,A -85,B 0,C 180,E1 1624.716,E2 1624.716} C_VEL
LIN {X 0,Y 730.313,Z 663.19,A -85,B 0,C 180,E1 1627.395,E2 1627.395} C_VEL
LIN {X 0,Y 730.689,Z 663.19,A -85,B 0,C 180,E1 1633.834,E2 1633.834} C_VEL
LIN {X 0,Y 730.778,Z 663.19,A -85,B 0,C 180,E1 1641.327,E2 1641.327} C_VEL
LIN {X 0,Y 731.171,Z 663.19,A -85,B 0,C 180,E1 1649.212,E2 1649.212} C_VEL
LIN {X 0,Y 730.66,Z 663.19,A -85,B 0,C 180,E1 1656.963,E2 1656.963} C_VEL
LIN {X 0,Y 730.435,Z 663.19,A -85,B 0,C 180,E1 1664.256,E2 1664.256} C_VEL
LIN {X 0,Y 730.757,Z 663.19,A -85,B 0,C 180,E1 1672.254,E2 1672.254} C_VEL
LIN {X 0,Y 731.18,Z 664.903,A -85,B 0,C 180,E1 1675.569,E2 1675.569} C_VEL
LIN {X 0,Y 736.418,Z 678.896,A -85,B 0,C 180,E1 1676.009,E2 1676.009} C_VEL
LIN {X 0,Y 736.388,Z 762.733,A -85,B 0,C 180,E1 1677.304,E2 1677.304} C_VEL
LIN {X 0,Y 735.282,Z 832.102,A -85,B 0,C 180,E1 1679.522,E2 1679.522} C_VEL
LIN {X 0,Y 733.839,Z 899.457,A -85,B 0,C 180,E1 1682.954,E2 1682.954} C_VEL
LIN {X 0,Y 732.49,Z 959.752,A -85,B 0,C 180,E1 1687.481,E2 1687.481} C_VEL
LIN {X 0,Y 731.633,Z 1007.928,A -85,B 0,C 180,E1 1692.675,E2 1692.675} C_VEL
LIN {X 0,Y 731.069,Z 1041.423,A -85,B 0,C 180,E1 1698.029,E2 1698.029} C_VEL
LIN {X 0,Y 730.782,Z 1060.28,A -85,B 0,C 180,E1 1702.848,E2 1702.848} C_VEL
LIN {X 0,Y 730.826,Z 1068.732,A -85,B 0,C 180,E1 1707.027,E2 1707.027} C_VEL
LIN {X 0,Y 731.321,Z 1069.802,A -85,B 0,C 180,E1 1711.783,E2 1711.783} C_VEL
LIN {X 0,Y 731.394,Z 1060.279,A -85,B 0,C 180,E1 1717.146,E2 1717.146} C_VEL
LIN {X 0,Y 731.441,Z 1036.487,A -85,B 0,C 180,E1 1722.933,E2 1722.933} C_VEL
LIN {X 0,Y 731.908,Z 997.905,A -85,B 0,C 180,E1 1728.575,E2 1728.575} C_VEL
LIN {X 0,Y 732.888,Z 946.51,A -85,B 0,C 180,E1 1733.656,E2 1733.656} C_VEL
LIN {X 0,Y 734.216,Z 885.082,A -85,B 0,C 180,E1 1737.899,E2 1737.899} C_VEL
LIN {X 0,Y 735.576,Z 816.146,A -85,B 0,C 180,E1 1741.099,E2 1741.099} C_VEL
LIN {X 0,Y 736.584,Z 743.967,A -85,B 0,C 180,E1 1743.094,E2 1743.094} C_VEL
LIN {X 0,Y 734.766,Z 671.248,A -85,B 0,C 180,E1 1744.166,E2 1744.166} C_VEL
LIN {X 0,Y 731.556,Z 663.19,A -85,B 0,C 180,E1 1744.458,E2 1744.458} C_VEL
LIN {X 0,Y 731.037,Z 663.19,A -85,B 0,C 180,E1 1754.232,E2 1754.232} C_VEL
LIN {X 0,Y 730.921,Z 663.19,A -85,B 0,C 180,E1 1763.698,E2 1763.698} C_VEL
LIN {X 0,Y 731.073,Z 663.19,A -85,B 0,C 180,E1 1772.138,E2 1772.138} C_VEL
LIN {X 0,Y 730.767,Z 663.19,A -85,B 0,C 180,E1 1781.207,E2 1781.207} C_VEL
LIN {X 0,Y 731.076,Z 663.19,A -85,B 0,C 180,E1 1788.612,E2 1788.612} C_VEL
LIN {X 0,Y 731.349,Z 663.19,A -85,B 0,C 180,E1 1795.822,E2 1795.822} C_VEL
LIN {X 0,Y 730.842,Z 663.19,A -85,B 0,C 180,E1 1804.155,E2 1804.155} C_VEL
LIN {X 0,Y 731.026,Z 663.19,A -85,B 0,C 180,E1 1811.363,E2 1811.363} C_VEL
LIN {X 0,Y 730.988,Z 663.19,A -85,B 0,C 180,E1 1819.285,E2 1819.285} C_VEL
LIN {X 0,Y 731.04,Z 663.19,A -85,B 0,C 180,E1 1826.497,E2 1826.497} C_VEL
LIN {X 0,Y 730.69,Z 663.19,A -85,B 0,C 180,E1 1834.82,E2 1834.82} C_VEL
LIN {X 0,Y 730.764,Z 663.19,A -85,B 0,C 180,E1 1840.846,E2 1840.846} C_VEL
LIN {X 0,Y 730.944,Z 663.19,A -85,B 0,C 180,E1 1849.261,E2 1849.261} C_VEL
LIN {X 0,Y 731.357,Z 665.006,A -85,B 0,C 180,E1 1852.651,E2 1852.651} C_VEL
LIN {X 0,Y 736.234,Z 682.353,A -85,B 0,C 180,E1 1853.109,E2 1853.109} C_VEL
LIN {X 0,Y 736.257,Z 762.18,A -85,B 0,C 180,E1 1854.495,E2 1854.495} C_VEL
LIN {X 0,Y 735.062,Z 832.411,A -85,B 0,C 180,E1 1856.916,E2 1856.916} C_VEL
LIN {X 0,Y 733.684,Z 898.907,A -85,B 0,C 180,E1 1860.524,E2 1860.524} C_VEL
LIN {X 0,Y 732.521,Z 956.444,A -85,B 0,C 180,E1 1865.047,E2 1865.047} C_VEL
LIN {X 0,Y 731.752,Z 1003.309,A -85,B 0,C 180,E1 1870.361,E2 1870.361} C_VEL
LIN {X 0,Y 731.507,Z 1037.103,A -85,B 0,C 180,E1 1876.208,E2 1876.208} C_VEL
LIN {X 0,Y 731.664,Z 1056.036,A -85,B 0,C 180,E1 1882.258,E2 1882.258} C_VEL
LIN {X 0,Y 731.711,Z 1060.147,A -85,B 0,C 180,E1 1888.218,E2 1888.218} C_VEL
LIN {X 0,Y 731.513,Z 1050.121,A -85,B 0,C 180,E1 1894.16,E2 1894.16} C_VEL
LIN {X 0,Y 731.472,Z 1025.014,A -85,B 0,C 180,E1 1900.149,E2 1900.149} C_VEL
LIN {X 0,Y 731.884,Z 985.771,A -85,B 0,C 180,E1 1905.78,E2 1905.78} C_VEL
LIN {X 0,Y 732.901,Z 934.835,A -85,B 0,C 180,E1 1910.752,E2 1910.752} C_VEL
LIN {X 0,Y 734.269,Z 873.342,A -85,B 0,C 180,E1 1914.951,E2 1914.951} C_VEL
LIN {X 0,Y 735.615,Z 804.408,A -85,B 0,C 180,E1 1918.114,E2 1918.114} C_VEL
LIN {X 0,Y 736.49,Z 731.906,A -85,B 0,C 180,E1 1920.09,E2 1920.09} C_VEL
LIN {X 0,Y 735.081,Z 672.597,A -85,B 0,C 180,E1 1920.974,E2 1920.974} C_VEL
LIN {X 0,Y 730.925,Z 663.19,A -85,B 0,C 180,E1 1921.421,E2 1921.421} C_VEL
LIN {X 0,Y 730.24,Z 663.19,A -85,B 0,C 180,E1 1928.812,E2 1928.812} C_VEL
LIN {X 0,Y 730.834,Z 663.19,A -85,B 0,C 180,E1 1935.933,E2 1935.933} C_VEL
LIN {X 0,Y 730.766,Z 663.19,A -85,B 0,C 180,E1 1943.721,E2 1943.721} C_VEL
LIN {X 0,Y 730.72,Z 663.19,A -85,B 0,C 180,E1 1951.881,E2 1951.881} C_VEL
LIN {X 0,Y 731.04,Z 663.19,A -85,B 0,C 180,E1 1958.709,E2 1958.709} C_VEL
LIN {X 0,Y 731.339,Z 663.19,A -85,B 0,C 180,E1 1967.427,E2 1967.427} C_VEL
LIN {X 0,Y 731.672,Z 663.19,A -85,B 0,C 180,E1 1977.04,E2 1977.04} C_VEL
LIN {X 0,Y 731.276,Z 663.19,A -85,B 0,C 180,E1 1985.372,E2 1985.372} C_VEL
LIN {X 0,Y 730.313,Z 663.19,A -85,B 0,C 180,E1 1987.395,E2 1987.395} C_VEL
LIN {X 0,Y 722.508,Z 663.19,A -85,B 0,C 180,E1 1990.128,E2 1990.128} C_VEL
LIN {X 0,Y 722.203,Z 663.19,A -85,B 0,C 180,E1 1995.244,E2 1995.244} C_VEL
LIN {X 0,Y 722.641,Z 663.19,A -85,B 0,C 180,E1 2001.579,E2 2001.579} C_VEL
LIN {X 0,Y 723.006,Z 663.19,A -85,B 0,C 180,E1 2009.575,E2 2009.575} C_VEL
LIN {X 0,Y 722.724,Z 663.19,A -85,B 0,C 180,E1 2016.781,E2 2016.781} C_VEL
LIN {X 0,Y 722.643,Z 663.19,A -85,B 0,C 180,E1 2023.618,E2 2023.618} C_VEL
LIN {X 0,Y 722.824,Z 663.19,A -85,B 0,C 180,E1 2031.967,E2 2031.967} C_VEL
LIN {X 0,Y 722.911,Z 664.363,A -85,B 0,C 180,E1 2035.112,E2 2035.112} C_VEL
LIN {X 0,Y 729.784,Z 681.693,A -85,B 0,C 180,E1 2035.69,E2 2035.69} C_VEL
LIN {X 0,Y 729.594,Z 763.53,A -85,B 0,C 180,E1 2036.978,E2 2036.978} C_VEL
LIN {X 0,Y 728.226,Z 832.106,A -85,B 0,C 180,E1 2039.195,E2 2039.195} C_VEL
LIN {X 0,Y 726.444,Z 899.313,A -85,B 0,C 180,E1 2042.647,E2 2042.647} C_VEL
LIN {X 0,Y 724.822,Z 958.558,A -85,B 0,C 180,E1 2047.12,E2 2047.12} C_VEL
LIN {X 0,Y 723.72,Z 1005.427,A -85,B 0,C 180,E1 2052.156,E2 2052.156} C_VEL
LIN {X 0,Y 722.983,Z 1038.323,A -85,B 0,C 180,E1 2057.278,E2 2057.278} C_VEL
LIN {X 0,Y 722.952,Z 1056.481,A -85,B 0,C 180,E1 2061.557,E2 2061.557} C_VEL
LIN {X 0,Y 722.836,Z 1068.733,A -85,B 0,C 180,E1 2066.994,E2 2066.994} C_VEL
LIN {X 0,Y 723.304,Z 1069.802,A -85,B 0,C 180,E1 2071.802,E2 2071.802} C_VEL
LIN {X 0,Y 723.37,Z 1060.279,A -85,B 0,C 180,E1 2077.226,E2 2077.226} C_VEL
LIN {X 0,Y 723.444,Z 1036.768,A -85,B 0,C 180,E1 2083.023,E2 2083.023} C_VEL
LIN {X 0,Y 724.053,Z 999.235,A -85,B 0,C 180,E1 2088.626,E2 2088.626} C_VEL
LIN {X 0,Y 725.227,Z 948.697,A -85,B 0,C 180,E1 2093.735,E2 2093.735} C_VEL
LIN {X 0,Y 726.856,Z 887.157,A -85,B 0,C 180,E1 2098.08,E2 2098.08} C_VEL
LIN {X 0,Y 728.513,Z 819.186,A -85,B 0,C 180,E1 2101.32,E2 2101.32} C_VEL
LIN {X 0,Y 729.765,Z 747.454,A -85,B 0,C 180,E1 2103.376,E2 2103.376} C_VEL
LIN {X 0,Y 728.046,Z 673.614,A -85,B 0,C 180,E1 2104.498,E2 2104.498} C_VEL
LIN {X 0,Y 723.504,Z 663.19,A -85,B 0,C 180,E1 2104.949,E2 2104.949} C_VEL
LIN {X 0,Y 722.925,Z 663.19,A -85,B 0,C 180,E1 2115.287,E2 2115.287} C_VEL
LIN {X 0,Y 722.642,Z 663.19,A -85,B 0,C 180,E1 2124.703,E2 2124.703} C_VEL
LIN {X 0,Y 722.56,Z 663.19,A -85,B 0,C 180,E1 2133.138,E2 2133.138} C_VEL
LIN {X 0,Y 722.839,Z 663.19,A -85,B 0,C 180,E1 2140.993,E2 2140.993} C_VEL
LIN {X 0,Y 723.097,Z 663.19,A -85,B 0,C 180,E1 2148.485,E2 2148.485} C_VEL
LIN {X 0,Y 723.342,Z 663.19,A -85,B 0,C 180,E1 2155.775,E2 2155.775} C_VEL
LIN {X 0,Y 722.81,Z 663.19,A -85,B 0,C 180,E1 2164.202,E2 2164.202} C_VEL
LIN {X 0,Y 722.938,Z 663.19,A -85,B 0,C 180,E1 2171.491,E2 2171.491} C_VEL
LIN {X 0,Y 723.162,Z 663.19,A -85,B 0,C 180,E1 2178.971,E2 2178.971} C_VEL
LIN {X 0,Y 722.863,Z 663.19,A -85,B 0,C 180,E1 2186.93,E2 2186.93} C_VEL
LIN {X 0,Y 722.874,Z 663.19,A -85,B 0,C 180,E1 2194.043,E2 2194.043} C_VEL
LIN {X 0,Y 722.349,Z 663.19,A -85,B 0,C 180,E1 2201.819,E2 2201.819} C_VEL
LIN {X 0,Y 723.001,Z 663.19,A -85,B 0,C 180,E1 2208.648,E2 2208.648} C_VEL
LIN {X 0,Y 723.252,Z 665.149,A -85,B 0,C 180,E1 2212.213,E2 2212.213} C_VEL
LIN {X 0,Y 729.557,Z 682.584,A -85,B 0,C 180,E1 2212.76,E2 2212.76} C_VEL
LIN {X 0,Y 729.42,Z 763.06,A -85,B 0,C 180,E1 2214.176,E2 2214.176} C_VEL
LIN {X 0,Y 727.968,Z 833.454,A -85,B 0,C 180,E1 2216.641,E2 2216.641} C_VEL
LIN {X 0,Y 726.213,Z 900.589,A -85,B 0,C 180,E1 2220.343,E2 2220.343} C_VEL
LIN {X 0,Y 724.764,Z 958.596,A -85,B 0,C 180,E1 2225.013,E2 2225.013} C_VEL
LIN {X 0,Y 723.884,Z 1004.949,A -85,B 0,C 180,E1 2230.408,E2 2230.408} C_VEL
LIN {X 0,Y 723.607,Z 1038.299,A -85,B 0,C 180,E1 2236.36,E2 2236.36} C_VEL
LIN {X 0,Y 723.609,Z 1055.968,A -85,B 0,C 180,E1 2242.171,E2 2242.171} C_VEL
LIN {X 0,Y 723.692,Z 1060.157,A -85,B 0,C 180,E1 2248.199,E2 2248.199} C_VEL
LIN {X 0,Y 723.485,Z 1050.209,A -85,B 0,C 180,E1 2254.207,E2 2254.207} C_VEL
LIN {X 0,Y 723.491,Z 1025.211,A -85,B 0,C 180,E1 2260.262,E2 2260.262} C_VEL
LIN {X 0,Y 724.06,Z 987.323,A -85,B 0,C 180,E1 2265.808,E2 2265.808} C_VEL
LIN {X 0,Y 725.274,Z 935.643,A -85,B 0,C 180,E1 2270.949,E2 2270.949} C_VEL
LIN {X 0,Y 726.97,Z 874.016,A -85,B 0,C 180,E1 2275.22,E2 2275.22} C_VEL
LIN {X 0,Y 728.632,Z 805.76,A -85,B 0,C 180,E1 2278.398,E2 2278.398} C_VEL
LIN {X 0,Y 729.774,Z 733.348,A -85,B 0,C 180,E1 2280.409,E2 2280.409} C_VEL
LIN {X 0,Y 728.247,Z 675.146,A -85,B 0,C 180,E1 2281.308,E2 2281.308} C_VEL
LIN {X 0,Y 722.809,Z 663.19,A -85,B 0,C 180,E1 2281.766,E2 2281.766} C_VEL
LIN {X 0,Y 722.47,Z 663.19,A -85,B 0,C 180,E1 2288.256,E2 2288.256} C_VEL
LIN {X 0,Y 722.643,Z 663.19,A -85,B 0,C 180,E1 2296.382,E2 2296.382} C_VEL
LIN {X 0,Y 722.688,Z 663.19,A -85,B 0,C 180,E1 2303.885,E2 2303.885} C_VEL
LIN {X 0,Y 722.759,Z 663.19,A -85,B 0,C 180,E1 2311.818,E2 2311.818} C_VEL
LIN {X 0,Y 722.589,Z 663.19,A -85,B 0,C 180,E1 2319.736,E2 2319.736} C_VEL
LIN {X 0,Y 723.328,Z 663.19,A -85,B 0,C 180,E1 2327.285,E2 2327.285} C_VEL
LIN {X 0,Y 723.632,Z 663.19,A -85,B 0,C 180,E1 2337.007,E2 2337.007} C_VEL
LIN {X 0,Y 723.254,Z 663.19,A -85,B 0,C 180,E1 2345.432,E2 2345.432} C_VEL
LIN {X 0,Y 722.508,Z 663.19,A -85,B 0,C 180,E1 2350.128,E2 2350.128} C_VEL
LIN {X 0,Y 715.208,Z 663.19,A -85,B 0,C 180,E1 2352.904,E2 2352.904} C_VEL
LIN {X 0,Y 714.491,Z 663.19,A -85,B 0,C 180,E1 2361.838,E2 2361.838} C_VEL
LIN {X 0,Y 714.865,Z 663.19,A -85,B 0,C 180,E1 2369.946,E2 2369.946} C_VEL
LIN {X 0,Y 714.578,Z 663.19,A -85,B 0,C 180,E1 2377.27,E2 2377.27} C_VEL
LIN {X 0,Y 714.281,Z 663.19,A -85,B 0,C 180,E1 2384.668,E2 2384.668} C_VEL
LIN {X 0,Y 714.629,Z 663.19,A -85,B 0,C 180,E1 2392.789,E2 2392.789} C_VEL
LIN {X 0,Y 714.817,Z 664.544,A -85,B 0,C 180,E1 2394.66,E2 2394.66} C_VEL
LIN {X 0,Y 723.191,Z 683.829,A -85,B 0,C 180,E1 2395.358,E2 2395.358} C_VEL
LIN {X 0,Y 722.837,Z 764.915,A -85,B 0,C 180,E1 2396.662,E2 2396.662} C_VEL
LIN {X 0,Y 721.166,Z 834.255,A -85,B 0,C 180,E1 2398.949,E2 2398.949} C_VEL
LIN {X 0,Y 718.985,Z 901.796,A -85,B 0,C 180,E1 2402.506,E2 2402.506} C_VEL
LIN {X 0,Y 717.114,Z 960.708,A -85,B 0,C 180,E1 2407.06,E2 2407.06} C_VEL
LIN {X 0,Y 715.84,Z 1008.267,A -85,B 0,C 180,E1 2412.324,E2 2412.324} C_VEL
LIN {X 0,Y 715.051,Z 1041.244,A -85,B 0,C 180,E1 2417.72,E2 2417.72} C_VEL
LIN {X 0,Y 714.793,Z 1060.28,A -85,B 0,C 180,E1 2422.687,E2 2422.687} C_VEL
LIN {X 0,Y 714.852,Z 1068.733,A -85,B 0,C 180,E1 2426.96,E2 2426.96} C_VEL
LIN {X 0,Y 715.296,Z 1069.802,A -85,B 0,C 180,E1 2431.823,E2 2431.823} C_VEL
LIN {X 0,Y 715.355,Z 1060.279,A -85,B 0,C 180,E1 2437.307,E2 2437.307} C_VEL
LIN {X 0,Y 715.439,Z 1036.77,A -85,B 0,C 180,E1 2443.171,E2 2443.171} C_VEL
LIN {X 0,Y 716.13,Z 999.233,A -85,B 0,C 180,E1 2448.84,E2 2448.84} C_VEL
LIN {X 0,Y 717.622,Z 948.696,A -85,B 0,C 180,E1 2454.003,E2 2454.003} C_VEL
LIN {X 0,Y 719.572,Z 886.776,A -85,B 0,C 180,E1 2458.413,E2 2458.413} C_VEL
LIN {X 0,Y 721.605,Z 818.576,A -85,B 0,C 180,E1 2461.679,E2 2461.679} C_VEL
LIN {X 0,Y 723.134,Z 745.677,A -85,B 0,C 180,E1 2463.76,E2 2463.76} C_VEL
LIN {X 0,Y 721.812,Z 677.296,A -85,B 0,C 180,E1 2464.796,E2 2464.796} C_VEL
LIN {X 0,Y 715.405,Z 663.19,A -85,B 0,C 180,E1 2465.414,E2 2465.414} C_VEL
LIN {X 0,Y 714.923,Z 663.19,A -85,B 0,C 180,E1 2475.281,E2 2475.281} C_VEL
LIN {X 0,Y 714.609,Z 663.19,A -85,B 0,C 180,E1 2484.784,E2 2484.784} C_VEL
LIN {X 0,Y 714.698,Z 663.19,A -85,B 0,C 180,E1 2492.818,E2 2492.818} C_VEL
LIN {X 0,Y 714.871,Z 663.19,A -85,B 0,C 180,E1 2500.773,E2 2500.773} C_VEL
LIN {X 0,Y 715.126,Z 663.19,A -85,B 0,C 180,E1 2508.354,E2 2508.354} C_VEL
LIN {X 0,Y 714.741,Z 663.19,A -85,B 0,C 180,E1 2516.944,E2 2516.944} C_VEL
LIN {X 0,Y 714.792,Z 663.19,A -85,B 0,C 180,E1 2524.249,E2 2524.249} C_VEL
LIN {X 0,Y 714.882,Z 663.19,A -85,B 0,C 180,E1 2531.623,E2 2531.623} C_VEL
LIN {X 0,Y 714.982,Z 663.19,A -85,B 0,C 180,E1 2539.298,E2 2539.298} C_VEL
LIN {X 0,Y 714.78,Z 663.19,A -85,B 0,C 180,E1 2547.149,E2 2547.149} C_VEL
LIN {X 0,Y 714.592,Z 663.19,A -85,B 0,C 180,E1 2555.214,E2 2555.214} C_VEL
LIN {X 0,Y 714.315,Z 663.19,A -85,B 0,C 180,E1 2561.997,E2 2561.997} C_VEL
LIN {X 0,Y 714.837,Z 663.19,A -85,B 0,C 180,E1 2569.683,E2 2569.683} C_VEL
LIN {X 0,Y 715.022,Z 664.61,A -85,B 0,C 180,E1 2571.748,E2 2571.748} C_VEL
LIN {X 0,Y 722.979,Z 684.464,A -85,B 0,C 180,E1 2572.427,E2 2572.427} C_VEL
LIN {X 0,Y 722.628,Z 763.884,A -85,B 0,C 180,E1 2573.852,E2 2573.852} C_VEL
LIN {X 0,Y 720.895,Z 833.903,A -85,B 0,C 180,E1 2576.332,E2 2576.332} C_VEL
LIN {X 0,Y 718.859,Z 899.995,A -85,B 0,C 180,E1 2580.009,E2 2580.009} C_VEL
LIN {X 0,Y 716.999,Z 957.396,A -85,B 0,C 180,E1 2584.641,E2 2584.641} C_VEL
LIN {X 0,Y 715.859,Z 1002.188,A -85,B 0,C 180,E1 2589.819,E2 2589.819} C_VEL
LIN {X 0,Y 715.24,Z 1034.652,A -85,B 0,C 180,E1 2595.398,E2 2595.398} C_VEL
LIN {X 0,Y 715.006,Z 1053.361,A -85,B 0,C 180,E1 2600.847,E2 2600.847} C_VEL
LIN {X 0,Y 715.15,Z 1060.5,A -85,B 0,C 180,E1 2606.961,E2 2606.961} C_VEL
LIN {X 0,Y 715.578,Z 1053.415,A -85,B 0,C 180,E1 2613.037,E2 2613.037} C_VEL
LIN {X 0,Y 715.941,Z 1031.64,A -85,B 0,C 180,E1 2619.14,E2 2619.14} C_VEL
LIN {X 0,Y 716.371,Z 995.123,A -85,B 0,C 180,E1 2625.029,E2 2625.029} C_VEL
LIN {X 0,Y 717.567,Z 945.061,A -85,B 0,C 180,E1 2630.407,E2 2630.407} C_VEL
LIN {X 0,Y 719.354,Z 885.677,A -85,B 0,C 180,E1 2634.826,E2 2634.826} C_VEL
LIN {X 0,Y 721.188,Z 818.71,A -85,B 0,C 180,E1 2638.235,E2 2638.235} C_VEL
LIN {X 0,Y 722.667,Z 744.348,A -85,B 0,C 180,E1 2640.545,E2 2640.545} C_VEL
LIN {X 0,Y 721.731,Z 678.073,A -85,B 0,C 180,E1 2641.627,E2 2641.627} C_VEL
LIN {X 0,Y 714.669,Z 663.19,A -85,B 0,C 180,E1 2642.282,E2 2642.282} C_VEL
LIN {X 0,Y 714.113,Z 663.19,A -85,B 0,C 180,E1 2649.145,E2 2649.145} C_VEL
LIN {X 0,Y 714.647,Z 663.19,A -85,B 0,C 180,E1 2656.369,E2 2656.369} C_VEL
LIN {X 0,Y 714.408,Z 663.19,A -85,B 0,C 180,E1 2664.806,E2 2664.806} C_VEL
LIN {X 0,Y 714.791,Z 663.19,A -85,B 0,C 180,E1 2671.692,E2 2671.692} C_VEL
LIN {X 0,Y 714.686,Z 663.19,A -85,B 0,C 180,E1 2679.502,E2 2679.502} C_VEL
LIN {X 0,Y 715.358,Z 663.19,A -85,B 0,C 180,E1 2687.141,E2 2687.141} C_VEL
LIN {X 0,Y 715.591,Z 663.19,A -85,B 0,C 180,E1 2696.974,E2 2696.974} C_VEL
LIN {X 0,Y 715.202,Z 663.19,A -85,B 0,C 180,E1 2705.493,E2 2705.493} C_VEL
LIN {X 0,Y 715.208,Z 663.19,A -85,B 0,C 180,E1 2712.904,E2 2712.904} C_VEL
LIN {X 0,Y 706.129,Z 663.19,A -85,B 0,C 180,E1 2715.667,E2 2715.667} C_VEL
LIN {X 0,Y 706.385,Z 663.19,A -85,B 0,C 180,E1 2722.102,E2 2722.102} C_VEL
LIN {X 0,Y 706.764,Z 663.19,A -85,B 0,C 180,E1 2730.325,E2 2730.325} C_VEL
LIN {X 0,Y 706.452,Z 663.19,A -85,B 0,C 180,E1 2737.774,E2 2737.774} C_VEL
LIN {X 0,Y 706.375,Z 663.19,A -85,B 0,C 180,E1 2744.312,E2 2744.312} C_VEL
LIN {X 0,Y 706.647,Z 663.19,A -85,B 0,C 180,E1 2752.296,E2 2752.296} C_VEL
LIN {X 0,Y 706.808,Z 664.86,A -85,B 0,C 180,E1 2754.202,E2 2754.202} C_VEL
LIN {X 0,Y 716.608,Z 687.26,A -85,B 0,C 180,E1 2755.034,E2 2755.034} C_VEL
LIN {X 0,Y 716.045,Z 766.732,A -85,B 0,C 180,E1 2756.354,E2 2756.354} C_VEL
LIN {X 0,Y 714.132,Z 835.268,A -85,B 0,C 180,E1 2758.652,E2 2758.652} C_VEL
LIN {X 0,Y 711.662,Z 901.62,A -85,B 0,C 180,E1 2762.186,E2 2762.186} C_VEL
LIN {X 0,Y 709.44,Z 960.895,A -85,B 0,C 180,E1 2766.815,E2 2766.815} C_VEL
LIN {X 0,Y 707.965,Z 1008.13,A -85,B 0,C 180,E1 2772.103,E2 2772.103} C_VEL
LIN {X 0,Y 707.059,Z 1040.259,A -85,B 0,C 180,E1 2777.379,E2 2777.379} C_VEL
LIN {X 0,Y 706.848,Z 1058.417,A -85,B 0,C 180,E1 2781.985,E2 2781.985} C_VEL
LIN {X 0,Y 706.808,Z 1068.968,A -85,B 0,C 180,E1 2787.151,E2 2787.151} C_VEL
LIN {X 0,Y 707.28,Z 1069.802,A -85,B 0,C 180,E1 2791.843,E2 2791.843} C_VEL
LIN {X 0,Y 707.338,Z 1060.279,A -85,B 0,C 180,E1 2797.391,E2 2797.391} C_VEL
LIN {X 0,Y 707.453,Z 1036.771,A -85,B 0,C 180,E1 2803.322,E2 2803.322} C_VEL
LIN {X 0,Y 708.243,Z 999.231,A -85,B 0,C 180,E1 2809.058,E2 2809.058} C_VEL
LIN {X 0,Y 709.959,Z 948.696,A -85,B 0,C 180,E1 2814.278,E2 2814.278} C_VEL
LIN {X 0,Y 712.265,Z 886.772,A -85,B 0,C 180,E1 2818.731,E2 2818.731} C_VEL
LIN {X 0,Y 714.68,Z 818.233,A -85,B 0,C 180,E1 2822.036,E2 2822.036} C_VEL
LIN {X 0,Y 716.472,Z 745.679,A -85,B 0,C 180,E1 2824.116,E2 2824.116} C_VEL
LIN {X 0,Y 715.244,Z 680.234,A -85,B 0,C 180,E1 2825.127,E2 2825.127} C_VEL
LIN {X 0,Y 707.292,Z 663.19,A -85,B 0,C 180,E1 2825.834,E2 2825.834} C_VEL
LIN {X 0,Y 706.668,Z 663.19,A -85,B 0,C 180,E1 2835.961,E2 2835.961} C_VEL
LIN {X 0,Y 706.679,Z 663.19,A -85,B 0,C 180,E1 2843.781,E2 2843.781} C_VEL
LIN {X 0,Y 706.626,Z 663.19,A -85,B 0,C 180,E1 2852.948,E2 2852.948} C_VEL
LIN {X 0,Y 706.872,Z 663.19,A -85,B 0,C 180,E1 2860.546,E2 2860.546} C_VEL
LIN {X 0,Y 707.121,Z 663.19,A -85,B 0,C 180,E1 2868.221,E2 2868.221} C_VEL
LIN {X 0,Y 706.751,Z 663.19,A -85,B 0,C 180,E1 2876.909,E2 2876.909} C_VEL
LIN {X 0,Y 706.771,Z 663.19,A -85,B 0,C 180,E1 2884.297,E2 2884.297} C_VEL
LIN {X 0,Y 706.514,Z 663.19,A -85,B 0,C 180,E1 2892.423,E2 2892.423} C_VEL
LIN {X 0,Y 706.925,Z 663.19,A -85,B 0,C 180,E1 2899.424,E2 2899.424} C_VEL
LIN {X 0,Y 706.672,Z 663.19,A -85,B 0,C 180,E1 2907.487,E2 2907.487} C_VEL
LIN {X 0,Y 706.7,Z 663.19,A -85,B 0,C 180,E1 2914.674,E2 2914.674} C_VEL
LIN {X 0,Y 706.249,Z 663.19,A -85,B 0,C 180,E1 2922.203,E2 2922.203} C_VEL
LIN {X 0,Y 706.858,Z 663.19,A -85,B 0,C 180,E1 2929.644,E2 2929.644} C_VEL
LIN {X 0,Y 706.973,Z 664.723,A -85,B 0,C 180,E1 2931.288,E2 2931.288} C_VEL
LIN {X 0,Y 716.507,Z 687.668,A -85,B 0,C 180,E1 2932.108,E2 2932.108} C_VEL
LIN {X 0,Y 715.805,Z 766.142,A -85,B 0,C 180,E1 2933.558,E2 2933.558} C_VEL
LIN {X 0,Y 713.749,Z 836.487,A -85,B 0,C 180,E1 2936.114,E2 2936.114} C_VEL
LIN {X 0,Y 711.373,Z 902.789,A -85,B 0,C 180,E1 2939.893,E2 2939.893} C_VEL
LIN {X 0,Y 709.29,Z 960.318,A -85,B 0,C 180,E1 2944.685,E2 2944.685} C_VEL
LIN {X 0,Y 708.025,Z 1005.803,A -85,B 0,C 180,E1 2950.15,E2 2950.15} C_VEL
LIN {X 0,Y 707.538,Z 1038.004,A -85,B 0,C 180,E1 2956.047,E2 2956.047} C_VEL
LIN {X 0,Y 707.506,Z 1055.831,A -85,B 0,C 180,E1 2961.991,E2 2961.991} C_VEL
LIN {X 0,Y 707.683,Z 1060.176,A -85,B 0,C 180,E1 2968.158,E2 2968.158} C_VEL
LIN {X 0,Y 707.467,Z 1050.386,A -85,B 0,C 180,E1 2974.302,E2 2974.302} C_VEL
LIN {X 0,Y 707.625,Z 1027.475,A -85,B 0,C 180,E1 2980.131,E2 2980.131} C_VEL
LIN {X 0,Y 708.395,Z 990.608,A -85,B 0,C 180,E1 2985.838,E2 2985.838} C_VEL
LIN {X 0,Y 709.981,Z 939.857,A -85,B 0,C 180,E1 2991.131,E2 2991.131} C_VEL
LIN {X 0,Y 712.288,Z 877.705,A -85,B 0,C 180,E1 2995.627,E2 2995.627} C_VEL
LIN {X 0,Y 714.671,Z 809.206,A -85,B 0,C 180,E1 2998.951,E2 2998.951} C_VEL
LIN {X 0,Y 716.317,Z 737.441,A -85,B 0,C 180,E1 3001.043,E2 3001.043} C_VEL
LIN {X 0,Y 715.027,Z 680.966,A -85,B 0,C 180,E1 3001.965,E2 3001.965} C_VEL
LIN {X 0,Y 706.602,Z 663.19,A -85,B 0,C 180,E1 3002.719,E2 3002.719} C_VEL
LIN {X 0,Y 706.06,Z 663.19,A -85,B 0,C 180,E1 3009.314,E2 3009.314} C_VEL
LIN {X 0,Y 706.732,Z 663.19,A -85,B 0,C 180,E1 3015.955,E2 3015.955} C_VEL
LIN {X 0,Y 706.592,Z 663.19,A -85,B 0,C 180,E1 3023.809,E2 3023.809} C_VEL
LIN {X 0,Y 706.782,Z 663.19,A -85,B 0,C 180,E1 3031.122,E2 3031.122} C_VEL
LIN {X 0,Y 706.722,Z 663.19,A -85,B 0,C 180,E1 3039.26,E2 3039.26} C_VEL
LIN {X 0,Y 707.404,Z 663.19,A -85,B 0,C 180,E1 3048.253,E2 3048.253} C_VEL
LIN {X 0,Y 707.059,Z 663.19,A -85,B 0,C 180,E1 3058.168,E2 3058.168} C_VEL
LIN {X 0,Y 707.176,Z 663.19,A -85,B 0,C 180,E1 3065.556,E2 3065.556} C_VEL
LIN {X 0,Y 707.123,Z 663.19,A -85,B 0,C 180,E1 3073.039,E2 3073.039} C_VEL
LIN {X 0,Y 706.129,Z 663.19,A -85,B 0,C 180,E1 3075.667,E2 3075.667} C_VEL
LIN {X 0,Y 698.55,Z 663.19,A -85,B 0,C 180,E1 3078.491,E2 3078.491} C_VEL
LIN {X 0,Y 698.818,Z 663.19,A -85,B 0,C 180,E1 3087.853,E2 3087.853} C_VEL
LIN {X 0,Y 698.94,Z 663.19,A -85,B 0,C 180,E1 3095.552,E2 3095.552} C_VEL
LIN {X 0,Y 698.625,Z 663.19,A -85,B 0,C 180,E1 3103.353,E2 3103.353} C_VEL
LIN {X 0,Y 698.612,Z 663.19,A -85,B 0,C 180,E1 3112.488,E2 3112.488} C_VEL
LIN {X 0,Y 698.729,Z 664.661,A -85,B 0,C 180,E1 3113.721,E2 3113.721} C_VEL
LIN {X 0,Y 710.048,Z 689.056,A -85,B 0,C 180,E1 3114.685,E2 3114.685} C_VEL
LIN {X 0,Y 709.327,Z 767.471,A -85,B 0,C 180,E1 3116.013,E2 3116.013} C_VEL
LIN {X 0,Y 707.079,Z 836.479,A -85,B 0,C 180,E1 3118.36,E2 3118.36} C_VEL
LIN {X 0,Y 704.244,Z 903.428,A -85,B 0,C 180,E1 3121.993,E2 3121.993} C_VEL
LIN {X 0,Y 701.743,Z 962.612,A -85,B 0,C 180,E1 3126.71,E2 3126.71} C_VEL
LIN {X 0,Y 700.078,Z 1009.232,A -85,B 0,C 180,E1 3132.044,E2 3132.044} C_VEL
LIN {X 0,Y 699.093,Z 1041.676,A -85,B 0,C 180,E1 3137.524,E2 3137.524} C_VEL
LIN {X 0,Y 698.838,Z 1060.281,A -85,B 0,C 180,E1 3142.519,E2 3142.519} C_VEL
LIN {X 0,Y 698.877,Z 1068.733,A -85,B 0,C 180,E1 3146.891,E2 3146.891} C_VEL
LIN {X 0,Y 699.282,Z 1069.802,A -85,B 0,C 180,E1 3151.864,E2 3151.864} C_VEL
LIN {X 0,Y 699.288,Z 1060.279,A -85,B 0,C 180,E1 3157.476,E2 3157.476} C_VEL
LIN {X 0,Y 699.449,Z 1036.772,A -85,B 0,C 180,E1 3163.478,E2 3163.478} C_VEL
LIN {X 0,Y 700.385,Z 1000.136,A -85,B 0,C 180,E1 3169.168,E2 3169.168} C_VEL
LIN {X 0,Y 702.354,Z 949.218,A -85,B 0,C 180,E1 3174.512,E2 3174.512} C_VEL
LIN {X 0,Y 704.972,Z 886.981,A -85,B 0,C 180,E1 3179.043,E2 3179.043} C_VEL
LIN {X 0,Y 707.772,Z 818.538,A -85,B 0,C 180,E1 3182.374,E2 3182.374} C_VEL
LIN {X 0,Y 709.781,Z 747.403,A -85,B 0,C 180,E1 3184.446,E2 3184.446} C_VEL
LIN {X 0,Y 708.502,Z 682.521,A -85,B 0,C 180,E1 3185.483,E2 3185.483} C_VEL
LIN {X 0,Y 699.112,Z 663.19,A -85,B 0,C 180,E1 3186.385,E2 3186.385} C_VEL
LIN {X 0,Y 698.732,Z 663.19,A -85,B 0,C 180,E1 3195.073,E2 3195.073} C_VEL
LIN {X 0,Y 698.462,Z 663.19,A -85,B 0,C 180,E1 3204.824,E2 3204.824} C_VEL
LIN {X 0,Y 698.777,Z 663.19,A -85,B 0,C 180,E1 3212.145,E2 3212.145} C_VEL
LIN {X 0,Y 698.814,Z 663.19,A -85,B 0,C 180,E1 3220.725,E2 3220.725} C_VEL
LIN {X 0,Y 698.705,Z 663.19,A -85,B 0,C 180,E1 3229.346,E2 3229.346} C_VEL
LIN {X 0,Y 698.771,Z 663.19,A -85,B 0,C 180,E1 3236.874,E2 3236.874} C_VEL
LIN {X 0,Y 698.741,Z 663.19,A -85,B 0,C 180,E1 3244.347,E2 3244.347} C_VEL
LIN {X 0,Y 698.73,Z 663.19,A -85,B 0,C 180,E1 3251.895,E2 3251.895} C_VEL
LIN {X 0,Y 698.811,Z 663.19,A -85,B 0,C 180,E1 3259.659,E2 3259.659} C_VEL
LIN {X 0,Y 698.56,Z 663.19,A -85,B 0,C 180,E1 3267.833,E2 3267.833} C_VEL
LIN {X 0,Y 698.523,Z 663.19,A -85,B 0,C 180,E1 3275.503,E2 3275.503} C_VEL
LIN {X 0,Y 698.428,Z 663.19,A -85,B 0,C 180,E1 3281.496,E2 3281.496} C_VEL
LIN {X 0,Y 698.919,Z 663.19,A -85,B 0,C 180,E1 3288.567,E2 3288.567} C_VEL
LIN {X 0,Y 699.011,Z 664.99,A -85,B 0,C 180,E1 3290.822,E2 3290.822} C_VEL
LIN {X 0,Y 709.964,Z 689.508,A -85,B 0,C 180,E1 3291.762,E2 3291.762} C_VEL
LIN {X 0,Y 709.061,Z 766.93,A -85,B 0,C 180,E1 3293.22,E2 3293.22} C_VEL
LIN {X 0,Y 706.722,Z 836.988,A -85,B 0,C 180,E1 3295.796,E2 3295.796} C_VEL
LIN {X 0,Y 703.981,Z 902.841,A -85,B 0,C 180,E1 3299.588,E2 3299.588} C_VEL
LIN {X 0,Y 701.536,Z 960.495,A -85,B 0,C 180,E1 3304.444,E2 3304.444} C_VEL
LIN {X 0,Y 700.101,Z 1006.473,A -85,B 0,C 180,E1 3310.053,E2 3310.053} C_VEL
LIN {X 0,Y 699.64,Z 1039.208,A -85,B 0,C 180,E1 3316.207,E2 3316.207} C_VEL
LIN {X 0,Y 699.356,Z 1056.912,A -85,B 0,C 180,E1 3322.524,E2 3322.524} C_VEL
LIN {X 0,Y 699.676,Z 1060.185,A -85,B 0,C 180,E1 3328.137,E2 3328.137} C_VEL
LIN {X 0,Y 699.438,Z 1050.474,A -85,B 0,C 180,E1 3334.352,E2 3334.352} C_VEL
LIN {X 0,Y 699.636,Z 1027.399,A -85,B 0,C 180,E1 3340.3,E2 3340.3} C_VEL
LIN {X 0,Y 700.503,Z 989.622,A -85,B 0,C 180,E1 3346.183,E2 3346.183} C_VEL
LIN {X 0,Y 702.386,Z 938.724,A -85,B 0,C 180,E1 3351.51,E2 3351.51} C_VEL
LIN {X 0,Y 705.04,Z 877.597,A -85,B 0,C 180,E1 3355.956,E2 3355.956} C_VEL
LIN {X 0,Y 707.771,Z 808.697,A -85,B 0,C 180,E1 3359.323,E2 3359.323} C_VEL
LIN {X 0,Y 709.747,Z 735.837,A -85,B 0,C 180,E1 3361.437,E2 3361.437} C_VEL
LIN {X 0,Y 708.507,Z 683.701,A -85,B 0,C 180,E1 3362.302,E2 3362.302} C_VEL
LIN {X 0,Y 698.607,Z 663.19,A -85,B 0,C 180,E1 3363.258,E2 3363.258} C_VEL
LIN {X 0,Y 697.953,Z 663.19,A -85,B 0,C 180,E1 3369.861,E2 3369.861} C_VEL
LIN {X 0,Y 698.44,Z 663.19,A -85,B 0,C 180,E1 3376.82,E2 3376.82} C_VEL
LIN {X 0,Y 698.33,Z 663.19,A -85,B 0,C 180,E1 3384.849,E2 3384.849} C_VEL
LIN {X 0,Y 698.557,Z 663.19,A -85,B 0,C 180,E1 3392.166,E2 3392.166} C_VEL
LIN {X 0,Y 698.783,Z 663.19,A -85,B 0,C 180,E1 3399.013,E2 3399.013} C_VEL
LIN {X 0,Y 699.414,Z 663.19,A -85,B 0,C 180,E1 3408.116,E2 3408.116} C_VEL
LIN {X 0,Y 699.081,Z 663.19,A -85,B 0,C 180,E1 3418.147,E2 3418.147} C_VEL
LIN {X 0,Y 699.123,Z 663.19,A -85,B 0,C 180,E1 3425.62,E2 3425.62} C_VEL
LIN {X 0,Y 699.019,Z 663.19,A -85,B 0,C 180,E1 3433.192,E2 3433.192} C_VEL
LIN {X 0,Y 698.55,Z 663.19,A -85,B 0,C 180,E1 3438.491,E2 3438.491} C_VEL
LIN {X 0,Y 690.621,Z 663.19,A -85,B 0,C 180,E1 3441.352,E2 3441.352} C_VEL
LIN {X 0,Y 690.798,Z 663.19,A -85,B 0,C 180,E1 3449.879,E2 3449.879} C_VEL
LIN {X 0,Y 690.57,Z 663.19,A -85,B 0,C 180,E1 3457.204,E2 3457.204} C_VEL
LIN {X 0,Y 690.266,Z 663.19,A -85,B 0,C 180,E1 3464.441,E2 3464.441} C_VEL
LIN {X 0,Y 690.576,Z 663.19,A -85,B 0,C 180,E1 3472.853,E2 3472.853} C_VEL
LIN {X 0,Y 690.927,Z 665.563,A -85,B 0,C 180,E1 3473.256,E2 3473.256} C_VEL
LIN {X 0,Y 703.493,Z 693.753,A -85,B 0,C 180,E1 3474.364,E2 3474.364} C_VEL
LIN {X 0,Y 702.506,Z 770.837,A -85,B 0,C 180,E1 3475.733,E2 3475.733} C_VEL
LIN {X 0,Y 700.015,Z 838.835,A -85,B 0,C 180,E1 3478.117,E2 3478.117} C_VEL
LIN {X 0,Y 696.803,Z 906.037,A -85,B 0,C 180,E1 3481.849,E2 3481.849} C_VEL
LIN {X 0,Y 694.018,Z 965.452,A -85,B 0,C 180,E1 3486.711,E2 3486.711} C_VEL
LIN {X 0,Y 692.188,Z 1010.945,A -85,B 0,C 180,E1 3492.072,E2 3492.072} C_VEL
LIN {X 0,Y 691.183,Z 1043.675,A -85,B 0,C 180,E1 3497.802,E2 3497.802} C_VEL
LIN {X 0,Y 690.849,Z 1061.848,A -85,B 0,C 180,E1 3503.066,E2 3503.066} C_VEL
LIN {X 0,Y 690.676,Z 1069.803,A -85,B 0,C 180,E1 3508.113,E2 3508.113} C_VEL
LIN {X 0,Y 690.866,Z 1068.733,A -85,B 0,C 180,E1 3513.146,E2 3513.146} C_VEL
LIN {X 0,Y 690.943,Z 1057.403,A -85,B 0,C 180,E1 3518.535,E2 3518.535} C_VEL
LIN {X 0,Y 691.429,Z 1035.075,A -85,B 0,C 180,E1 3523.96,E2 3523.96} C_VEL
LIN {X 0,Y 692.586,Z 998.664,A -85,B 0,C 180,E1 3529.576,E2 3529.576} C_VEL
LIN {X 0,Y 694.836,Z 947.609,A -85,B 0,C 180,E1 3534.939,E2 3534.939} C_VEL
LIN {X 0,Y 697.85,Z 885.439,A -85,B 0,C 180,E1 3539.467,E2 3539.467} C_VEL
LIN {X 0,Y 700.939,Z 817.077,A -85,B 0,C 180,E1 3542.788,E2 3542.788} C_VEL
LIN {X 0,Y 703.236,Z 745.681,A -85,B 0,C 180,E1 3544.85,E2 3544.85} C_VEL
LIN {X 0,Y 702.105,Z 685.735,A -85,B 0,C 180,E1 3545.816,E2 3545.816} C_VEL
LIN {X 0,Y 690.932,Z 663.19,A -85,B 0,C 180,E1 3546.884,E2 3546.884} C_VEL
LIN {X 0,Y 690.4,Z 663.19,A -85,B 0,C 180,E1 3556.153,E2 3556.153} C_VEL
LIN {X 0,Y 690.517,Z 663.19,A -85,B 0,C 180,E1 3564.358,E2 3564.358} C_VEL
LIN {X 0,Y 690.411,Z 663.19,A -85,B 0,C 180,E1 3573.198,E2 3573.198} C_VEL
LIN {X 0,Y 690.578,Z 663.19,A -85,B 0,C 180,E1 3581.402,E2 3581.402} C_VEL
LIN {X 0,Y 690.73,Z 663.19,A -85,B 0,C 180,E1 3589.221,E2 3589.221} C_VEL
LIN {X 0,Y 690.803,Z 663.19,A -85,B 0,C 180,E1 3596.838,E2 3596.838} C_VEL
LIN {X 0,Y 690.735,Z 663.19,A -85,B 0,C 180,E1 3604.397,E2 3604.397} C_VEL
LIN {X 0,Y 690.554,Z 663.19,A -85,B 0,C 180,E1 3612.259,E2 3612.259} C_VEL
LIN {X 0,Y 690.707,Z 663.19,A -85,B 0,C 180,E1 3619.899,E2 3619.899} C_VEL
LIN {X 0,Y 690.476,Z 663.19,A -85,B 0,C 180,E1 3628.188,E2 3628.188} C_VEL
LIN {X 0,Y 690.51,Z 663.19,A -85,B 0,C 180,E1 3635.609,E2 3635.609} C_VEL
LIN {X 0,Y 690.125,Z 663.19,A -85,B 0,C 180,E1 3642.6,E2 3642.6} C_VEL
LIN {X 0,Y 690.992,Z 664.82,A -85,B 0,C 180,E1 3650.332,E2 3650.332} C_VEL
LIN {X 0,Y 703.491,Z 693.076,A -85,B 0,C 180,E1 3651.433,E2 3651.433} C_VEL
LIN {X 0,Y 702.303,Z 769.625,A -85,B 0,C 180,E1 3652.928,E2 3652.928} C_VEL
LIN {X 0,Y 699.582,Z 840.345,A -85,B 0,C 180,E1 3655.604,E2 3655.604} C_VEL
LIN {X 0,Y 696.468,Z 906.167,A -85,B 0,C 180,E1 3659.515,E2 3659.515} C_VEL
LIN {X 0,Y 693.829,Z 963.416,A -85,B 0,C 180,E1 3664.486,E2 3664.486} C_VEL
LIN {X 0,Y 692.252,Z 1008.435,A -85,B 0,C 180,E1 3670.151,E2 3670.151} C_VEL
LIN {X 0,Y 691.715,Z 1040.332,A -85,B 0,C 180,E1 3676.369,E2 3676.369} C_VEL
LIN {X 0,Y 691.366,Z 1056.863,A -85,B 0,C 180,E1 3682.438,E2 3682.438} C_VEL
LIN {X 0,Y 691.655,Z 1060.195,A -85,B 0,C 180,E1 3688.115,E2 3688.115} C_VEL
LIN {X 0,Y 691.44,Z 1050.563,A -85,B 0,C 180,E1 3694.402,E2 3694.402} C_VEL
LIN {X 0,Y 691.626,Z 1027.576,A -85,B 0,C 180,E1 3700.421,E2 3700.421} C_VEL
LIN {X 0,Y 692.659,Z 991.173,A -85,B 0,C 180,E1 3706.208,E2 3706.208} C_VEL
LIN {X 0,Y 694.736,Z 941.05,A -85,B 0,C 180,E1 3711.59,E2 3711.59} C_VEL
LIN {X 0,Y 697.724,Z 879.816,A -85,B 0,C 180,E1 3716.147,E2 3716.147} C_VEL
LIN {X 0,Y 700.772,Z 811.359,A -85,B 0,C 180,E1 3719.571,E2 3719.571} C_VEL
LIN {X 0,Y 703.031,Z 738.411,A -85,B 0,C 180,E1 3721.755,E2 3721.755} C_VEL
LIN {X 0,Y 701.963,Z 686.72,A -85,B 0,C 180,E1 3722.644,E2 3722.644} C_VEL
LIN {X 0,Y 690.58,Z 663.19,A -85,B 0,C 180,E1 3723.808,E2 3723.808} C_VEL
LIN {X 0,Y 689.874,Z 663.19,A -85,B 0,C 180,E1 3730.642,E2 3730.642} C_VEL
LIN {X 0,Y 690.201,Z 663.19,A -85,B 0,C 180,E1 3737.897,E2 3737.897} C_VEL
LIN {X 0,Y 690.204,Z 663.19,A -85,B 0,C 180,E1 3745.476,E2 3745.476} C_VEL
LIN {X 0,Y 690.314,Z 663.19,A -85,B 0,C 180,E1 3753.225,E2 3753.225} C_VEL
LIN {X 0,Y 690.45,Z 663.19,A -85,B 0,C 180,E1 3760.093,E2 3760.093} C_VEL
LIN {X 0,Y 691.389,Z 663.19,A -85,B 0,C 180,E1 3767.977,E2 3767.977} C_VEL
LIN {X 0,Y 691.085,Z 663.19,A -85,B 0,C 180,E1 3778.126,E2 3778.126} C_VEL
LIN {X 0,Y 691.094,Z 663.19,A -85,B 0,C 180,E1 3785.685,E2 3785.685} C_VEL
LIN {X 0,Y 690.927,Z 663.19,A -85,B 0,C 180,E1 3793.35,E2 3793.35} C_VEL
LIN {X 0,Y 690.621,Z 663.19,A -85,B 0,C 180,E1 3801.352,E2 3801.352} C_VEL
LIN {X 0,Y 681.915,Z 663.19,A -85,B 0,C 180,E1 3804.225,E2 3804.225} C_VEL
LIN {X 0,Y 682.674,Z 663.19,A -85,B 0,C 180,E1 3811.515,E2 3811.515} C_VEL
LIN {X 0,Y 682.363,Z 663.19,A -85,B 0,C 180,E1 3819.358,E2 3819.358} C_VEL
LIN {X 0,Y 682.053,Z 663.19,A -85,B 0,C 180,E1 3826.342,E2 3826.342} C_VEL
LIN {X 0,Y 682.727,Z 664.755,A -85,B 0,C 180,E1 3832.73,E2 3832.73} C_VEL
LIN {X 0,Y 696.984,Z 696.294,A -85,B 0,C 180,E1 3834.011,E2 3834.011} C_VEL
LIN {X 0,Y 695.778,Z 772.436,A -85,B 0,C 180,E1 3835.401,E2 3835.401} C_VEL
LIN {X 0,Y 692.978,Z 840.98,A -85,B 0,C 180,E1 3837.858,E2 3837.858} C_VEL
LIN {X 0,Y 689.436,Z 907.444,A -85,B 0,C 180,E1 3841.622,E2 3841.622} C_VEL
LIN {X 0,Y 686.349,Z 966.582,A -85,B 0,C 180,E1 3846.547,E2 3846.547} C_VEL
LIN {X 0,Y 684.328,Z 1011.397,A -85,B 0,C 180,E1 3851.927,E2 3851.927} C_VEL
LIN {X 0,Y 683.197,Z 1043.675,A -85,B 0,C 180,E1 3857.657,E2 3857.657} C_VEL
LIN {X 0,Y 682.847,Z 1061.848,A -85,B 0,C 180,E1 3862.985,E2 3862.985} C_VEL
LIN {X 0,Y 682.678,Z 1069.803,A -85,B 0,C 180,E1 3868.091,E2 3868.091} C_VEL
LIN {X 0,Y 682.864,Z 1068.733,A -85,B 0,C 180,E1 3873.183,E2 3873.183} C_VEL
LIN {X 0,Y 682.982,Z 1057.979,A -85,B 0,C 180,E1 3878.443,E2 3878.443} C_VEL
LIN {X 0,Y 683.463,Z 1035.074,A -85,B 0,C 180,E1 3884.127,E2 3884.127} C_VEL
LIN {X 0,Y 684.768,Z 999.064,A -85,B 0,C 180,E1 3889.758,E2 3889.758} C_VEL
LIN {X 0,Y 687.228,Z 949.086,A -85,B 0,C 180,E1 3895.1,E2 3895.1} C_VEL
LIN {X 0,Y 690.575,Z 886.685,A -85,B 0,C 180,E1 3899.728,E2 3899.728} C_VEL
LIN {X 0,Y 694.047,Z 818.246,A -85,B 0,C 180,E1 3903.108,E2 3903.108} C_VEL
LIN {X 0,Y 696.612,Z 747.381,A -85,B 0,C 180,E1 3905.193,E2 3905.193} C_VEL
LIN {X 0,Y 695.653,Z 688.692,A -85,B 0,C 180,E1 3906.164,E2 3906.164} C_VEL
LIN {X 0,Y 682.742,Z 663.19,A -85,B 0,C 180,E1 3907.348,E2 3907.348} C_VEL
LIN {X 0,Y 682.36,Z 663.19,A -85,B 0,C 180,E1 3916.241,E2 3916.241} C_VEL
LIN {X 0,Y 682.544,Z 663.19,A -85,B 0,C 180,E1 3924.187,E2 3924.187} C_VEL
LIN {X 0,Y 682.523,Z 663.19,A -85,B 0,C 180,E1 3932.863,E2 3932.863} C_VEL
LIN {X 0,Y 682.594,Z 663.19,A -85,B 0,C 180,E1 3941.176,E2 3941.176} C_VEL
LIN {X 0,Y 682.754,Z 663.19,A -85,B 0,C 180,E1 3949.094,E2 3949.094} C_VEL
LIN {X 0,Y 682.813,Z 663.19,A -85,B 0,C 180,E1 3956.801,E2 3956.801} C_VEL
LIN {X 0,Y 682.705,Z 663.19,A -85,B 0,C 180,E1 3964.449,E2 3964.449} C_VEL
LIN {X 0,Y 682.591,Z 663.19,A -85,B 0,C 180,E1 3972.181,E2 3972.181} C_VEL
LIN {X 0,Y 682.639,Z 663.19,A -85,B 0,C 180,E1 3980.144,E2 3980.144} C_VEL
LIN {X 0,Y 682.406,Z 663.19,A -85,B 0,C 180,E1 3988.552,E2 3988.552} C_VEL
LIN {X 0,Y 682.488,Z 663.19,A -85,B 0,C 180,E1 3996.093,E2 3996.093} C_VEL
LIN {X 0,Y 682.051,Z 663.19,A -85,B 0,C 180,E1 4003.732,E2 4003.732} C_VEL
LIN {X 0,Y 683.021,Z 665.105,A -85,B 0,C 180,E1 4009.837,E2 4009.837} C_VEL
LIN {X 0,Y 696.964,Z 695.072,A -85,B 0,C 180,E1 4011.074,E2 4011.074} C_VEL
LIN {X 0,Y 695.529,Z 772.029,A -85,B 0,C 180,E1 4012.619,E2 4012.619} C_VEL
LIN {X 0,Y 692.446,Z 842.86,A -85,B 0,C 180,E1 4015.373,E2 4015.373} C_VEL
LIN {X 0,Y 689.039,Z 907.507,A -85,B 0,C 180,E1 4019.297,E2 4019.297} C_VEL
LIN {X 0,Y 686.098,Z 964.694,A -85,B 0,C 180,E1 4024.356,E2 4024.356} C_VEL
LIN {X 0,Y 684.282,Z 1008.175,A -85,B 0,C 180,E1 4029.91,E2 4029.91} C_VEL
LIN {X 0,Y 683.676,Z 1040.199,A -85,B 0,C 180,E1 4036.205,E2 4036.205} C_VEL
LIN {X 0,Y 683.384,Z 1056.814,A -85,B 0,C 180,E1 4042.349,E2 4042.349} C_VEL
LIN {X 0,Y 683.637,Z 1060.204,A -85,B 0,C 180,E1 4048.093,E2 4048.093} C_VEL
LIN {X 0,Y 683.412,Z 1050.651,A -85,B 0,C 180,E1 4054.454,E2 4054.454} C_VEL
LIN {X 0,Y 683.643,Z 1027.753,A -85,B 0,C 180,E1 4060.544,E2 4060.544} C_VEL
LIN {X 0,Y 684.797,Z 991.455,A -85,B 0,C 180,E1 4066.399,E2 4066.399} C_VEL
LIN {X 0,Y 687.125,Z 941.925,A -85,B 0,C 180,E1 4071.802,E2 4071.802} C_VEL
LIN {X 0,Y 690.455,Z 881.022,A -85,B 0,C 180,E1 4076.406,E2 4076.406} C_VEL
LIN {X 0,Y 693.815,Z 813.144,A -85,B 0,C 180,E1 4079.862,E2 4079.862} C_VEL
LIN {X 0,Y 696.327,Z 740.665,A -85,B 0,C 180,E1 4082.085,E2 4082.085} C_VEL
LIN {X 0,Y 695.409,Z 689.545,A -85,B 0,C 180,E1 4082.998,E2 4082.998} C_VEL
LIN {X 0,Y 682.579,Z 663.19,A -85,B 0,C 180,E1 4084.251,E2 4084.251} C_VEL
LIN {X 0,Y 682.18,Z 663.19,A -85,B 0,C 180,E1 4092.686,E2 4092.686} C_VEL
LIN {X 0,Y 682.316,Z 663.19,A -85,B 0,C 180,E1 4100.674,E2 4100.674} C_VEL
LIN {X 0,Y 682.58,Z 663.19,A -85,B 0,C 180,E1 4108.794,E2 4108.794} C_VEL
LIN {X 0,Y 682.833,Z 663.19,A -85,B 0,C 180,E1 4117.163,E2 4117.163} C_VEL
LIN {X 0,Y 683.294,Z 663.19,A -85,B 0,C 180,E1 4126.527,E2 4126.527} C_VEL
LIN {X 0,Y 682.293,Z 663.19,A -85,B 0,C 180,E1 4134.269,E2 4134.269} C_VEL
LIN {X 0,Y 682.521,Z 663.19,A -85,B 0,C 180,E1 4139.377,E2 4139.377} C_VEL
LIN {X 0,Y 683.043,Z 663.19,A -85,B 0,C 180,E1 4145.753,E2 4145.753} C_VEL
LIN {X 0,Y 682.834,Z 663.19,A -85,B 0,C 180,E1 4153.511,E2 4153.511} C_VEL
LIN {X 0,Y 682.531,Z 663.19,A -85,B 0,C 180,E1 4161.541,E2 4161.541} C_VEL
LIN {X 0,Y 681.915,Z 663.19,A -85,B 0,C 180,E1 4164.225,E2 4164.225} C_VEL
LIN {X 0,Y 674.485,Z 663.19,A -85,B 0,C 180,E1 4167.163,E2 4167.163} C_VEL
LIN {X 0,Y 674.869,Z 663.19,A -85,B 0,C 180,E1 4175.011,E2 4175.011} C_VEL
LIN {X 0,Y 674.531,Z 663.19,A -85,B 0,C 180,E1 4183.356,E2 4183.356} C_VEL
LIN {X 0,Y 674.791,Z 664.831,A -85,B 0,C 180,E1 4192.216,E2 4192.216} C_VEL
LIN {X 0,Y 690.515,Z 698.317,A -85,B 0,C 180,E1 4193.646,E2 4193.646} C_VEL
LIN {X 0,Y 689.122,Z 773.364,A -85,B 0,C 180,E1 4195.046,E2 4195.046} C_VEL
LIN {X 0,Y 685.976,Z 841.921,A -85,B 0,C 180,E1 4197.537,E2 4197.537} C_VEL
LIN {X 0,Y 682.108,Z 908.429,A -85,B 0,C 180,E1 4201.36,E2 4201.36} C_VEL
LIN {X 0,Y 678.733,Z 965.64,A -85,B 0,C 180,E1 4206.174,E2 4206.174} C_VEL
LIN {X 0,Y 676.517,Z 1011.399,A -85,B 0,C 180,E1 4211.711,E2 4211.711} C_VEL
LIN {X 0,Y 675.199,Z 1042.96,A -85,B 0,C 180,E1 4217.352,E2 4217.352} C_VEL
LIN {X 0,Y 674.92,Z 1060.307,A -85,B 0,C 180,E1 4222.264,E2 4222.264} C_VEL
LIN {X 0,Y 674.934,Z 1068.734,A -85,B 0,C 180,E1 4226.78,E2 4226.78} C_VEL
LIN {X 0,Y 675.283,Z 1069.803,A -85,B 0,C 180,E1 4231.931,E2 4231.931} C_VEL
LIN {X 0,Y 675.212,Z 1060.279,A -85,B 0,C 180,E1 4237.744,E2 4237.744} C_VEL
LIN {X 0,Y 675.581,Z 1038.326,A -85,B 0,C 180,E1 4243.632,E2 4243.632} C_VEL
LIN {X 0,Y 676.842,Z 1002.77,A -85,B 0,C 180,E1 4249.499,E2 4249.499} C_VEL
LIN {X 0,Y 679.47,Z 954.176,A -85,B 0,C 180,E1 4254.939,E2 4254.939} C_VEL
LIN {X 0,Y 683.038,Z 893.378,A -85,B 0,C 180,E1 4259.648,E2 4259.648} C_VEL
LIN {X 0,Y 686.897,Z 824.817,A -85,B 0,C 180,E1 4263.207,E2 4263.207} C_VEL
LIN {X 0,Y 689.742,Z 753.234,A -85,B 0,C 180,E1 4265.453,E2 4265.453} C_VEL
LIN {X 0,Y 689.066,Z 691.313,A -85,B 0,C 180,E1 4266.532,E2 4266.532} C_VEL
LIN {X 0,Y 674.506,Z 663.19,A -85,B 0,C 180,E1 4267.936,E2 4267.936} C_VEL
LIN {X 0,Y 674.236,Z 663.19,A -85,B 0,C 180,E1 4276.62,E2 4276.62} C_VEL
LIN {X 0,Y 674.302,Z 663.19,A -85,B 0,C 180,E1 4285.169,E2 4285.169} C_VEL
LIN {X 0,Y 674.554,Z 663.19,A -85,B 0,C 180,E1 4292.62,E2 4292.62} C_VEL
LIN {X 0,Y 674.656,Z 663.19,A -85,B 0,C 180,E1 4300.946,E2 4300.946} C_VEL
LIN {X 0,Y 674.772,Z 663.19,A -85,B 0,C 180,E1 4308.963,E2 4308.963} C_VEL
LIN {X 0,Y 674.822,Z 663.19,A -85,B 0,C 180,E1 4316.763,E2 4316.763} C_VEL
LIN {X 0,Y 674.69,Z 663.19,A -85,B 0,C 180,E1 4324.502,E2 4324.502} C_VEL
LIN {X 0,Y 674.55,Z 663.19,A -85,B 0,C 180,E1 4332.328,E2 4332.328} C_VEL
LIN {X 0,Y 674.555,Z 663.19,A -85,B 0,C 180,E1 4340.396,E2 4340.396} C_VEL
LIN {X 0,Y 674.614,Z 663.19,A -85,B 0,C 180,E1 4347.45,E2 4347.45} C_VEL
LIN {X 0,Y 674.574,Z 663.19,A -85,B 0,C 180,E1 4354.995,E2 4354.995} C_VEL
LIN {X 0,Y 674.096,Z 663.19,A -85,B 0,C 180,E1 4363.021,E2 4363.021} C_VEL
LIN {X 0,Y 674.863,Z 664.111,A -85,B 0,C 180,E1 4369.298,E2 4369.298} C_VEL
LIN {X 0,Y 690.476,Z 697.413,A -85,B 0,C 180,E1 4370.713,E2 4370.713} C_VEL
LIN {X 0,Y 688.866,Z 772.506,A -85,B 0,C 180,E1 4372.255,E2 4372.255} C_VEL
LIN {X 0,Y 685.546,Z 841.337,A -85,B 0,C 180,E1 4374.936,E2 4374.936} C_VEL
LIN {X 0,Y 681.725,Z 906.475,A -85,B 0,C 180,E1 4378.894,E2 4378.894} C_VEL
LIN {X 0,Y 678.345,Z 963.508,A -85,B 0,C 180,E1 4383.955,E2 4383.955} C_VEL
LIN {X 0,Y 676.396,Z 1007.917,A -85,B 0,C 180,E1 4389.666,E2 4389.666} C_VEL
LIN {X 0,Y 675.52,Z 1038.739,A -85,B 0,C 180,E1 4395.704,E2 4395.704} C_VEL
LIN {X 0,Y 675.377,Z 1056.76,A -85,B 0,C 180,E1 4402.257,E2 4402.257} C_VEL
LIN {X 0,Y 675.633,Z 1060.214,A -85,B 0,C 180,E1 4408.07,E2 4408.07} C_VEL
LIN {X 0,Y 675.402,Z 1050.74,A -85,B 0,C 180,E1 4414.507,E2 4414.507} C_VEL
LIN {X 0,Y 675.668,Z 1027.931,A -85,B 0,C 180,E1 4420.67,E2 4420.67} C_VEL
LIN {X 0,Y 676.956,Z 991.736,A -85,B 0,C 180,E1 4426.595,E2 4426.595} C_VEL
LIN {X 0,Y 679.567,Z 942.086,A -85,B 0,C 180,E1 4432.082,E2 4432.082} C_VEL
LIN {X 0,Y 683.26,Z 880.297,A -85,B 0,C 180,E1 4436.795,E2 4436.795} C_VEL
LIN {X 0,Y 687.032,Z 812.213,A -85,B 0,C 180,E1 4440.27,E2 4440.27} C_VEL
LIN {X 0,Y 689.795,Z 740.311,A -85,B 0,C 180,E1 4442.476,E2 4442.476} C_VEL
LIN {X 0,Y 688.928,Z 692.367,A -85,B 0,C 180,E1 4443.355,E2 4443.355} C_VEL
LIN {X 0,Y 674.625,Z 663.19,A -85,B 0,C 180,E1 4444.821,E2 4444.821} C_VEL
LIN {X 0,Y 674.317,Z 663.19,A -85,B 0,C 180,E1 4453.305,E2 4453.305} C_VEL
LIN {X 0,Y 674.459,Z 663.19,A -85,B 0,C 180,E1 4461.785,E2 4461.785} C_VEL
LIN {X 0,Y 674.646,Z 663.19,A -85,B 0,C 180,E1 4471.089,E2 4471.089} C_VEL
LIN {X 0,Y 674.519,Z 663.19,A -85,B 0,C 180,E1 4479.602,E2 4479.602} C_VEL
LIN {X 0,Y 675.378,Z 663.19,A -85,B 0,C 180,E1 4487.687,E2 4487.687} C_VEL
LIN {X 0,Y 675.114,Z 663.19,A -85,B 0,C 180,E1 4498.081,E2 4498.081} C_VEL
LIN {X 0,Y 675.025,Z 663.19,A -85,B 0,C 180,E1 4505.821,E2 4505.821} C_VEL
LIN {X 0,Y 674.747,Z 663.19,A -85,B 0,C 180,E1 4513.676,E2 4513.676} C_VEL
LIN {X 0,Y 674.425,Z 663.19,A -85,B 0,C 180,E1 4521.813,E2 4521.813} C_VEL
LIN {X 0,Y 674.485,Z 663.19,A -85,B 0,C 180,E1 4527.163,E2 4527.163} C_VEL
LIN {X 0,Y 674.554,Z 665.19,A -85,B 0,C 180,E1 4527.332,E2 4527.332} C_VEL
LIN {X 0,Y 674.554,Z 1070.125,A -85,B 0,C 180,E1 4527.332,E2 4527.332} C_VEL
LIN {X 0,Y 673.788,Z 1070.125,A -85,B 0,C 180,E1 4408.496,E2 4408.496} C_VEL
LIN {X 0,Y 675.51,Z 1068.125,A -85,B 0,C 180,E1 4408.409,E2 4408.409} C_VEL
LIN {X 0,Y 675.51,Z 1062.169,A -85,B 0,C 180,E1 4408.409,E2 4408.409} C_VEL
LIN {X 0,Y 675.57,Z 1060.169,A -85,B 0,C 180,E1 4408.236,E2 4408.236} C_VEL
LIN {X 0,Y 666.888,Z 1057.453,A -85,B 0,C 180,E1 4411.153,E2 4411.153} C_VEL
LIN {X 0,Y 666.977,Z 1045.25,A -85,B 0,C 180,E1 4416.527,E2 4416.527} C_VEL
LIN {X 0,Y 667.637,Z 1021.585,A -85,B 0,C 180,E1 4422.095,E2 4422.095} C_VEL
LIN {X 0,Y 669.254,Z 985.61,A -85,B 0,C 180,E1 4427.641,E2 4427.641} C_VEL
LIN {X 0,Y 672.302,Z 935.164,A -85,B 0,C 180,E1 4433.019,E2 4433.019} C_VEL
LIN {X 0,Y 676.52,Z 873.839,A -85,B 0,C 180,E1 4437.554,E2 4437.554} C_VEL
LIN {X 0,Y 680.567,Z 805.926,A -85,B 0,C 180,E1 4440.901,E2 4440.901} C_VEL
LIN {X 0,Y 683.544,Z 733.65,A -85,B 0,C 180,E1 4443.004,E2 4443.004} C_VEL
LIN {X 0,Y 682.409,Z 695.221,A -85,B 0,C 180,E1 4443.723,E2 4443.723} C_VEL
LIN {X 0,Y 666.58,Z 663.19,A -85,B 0,C 180,E1 4445.272,E2 4445.272} C_VEL
LIN {X 0,Y 666.393,Z 663.19,A -85,B 0,C 180,E1 4454.176,E2 4454.176} C_VEL
LIN {X 0,Y 666.505,Z 663.19,A -85,B 0,C 180,E1 4462.899,E2 4462.899} C_VEL
LIN {X 0,Y 666.631,Z 663.19,A -85,B 0,C 180,E1 4471.136,E2 4471.136} C_VEL
LIN {X 0,Y 666.579,Z 663.19,A -85,B 0,C 180,E1 4479.348,E2 4479.348} C_VEL
LIN {X 0,Y 667.385,Z 663.19,A -85,B 0,C 180,E1 4487.537,E2 4487.537} C_VEL
LIN {X 0,Y 667.117,Z 663.19,A -85,B 0,C 180,E1 4498.058,E2 4498.058} C_VEL
LIN {X 0,Y 666.976,Z 663.19,A -85,B 0,C 180,E1 4505.892,E2 4505.892} C_VEL
LIN {X 0,Y 666.664,Z 663.19,A -85,B 0,C 180,E1 4513.845,E2 4513.845} C_VEL
LIN {X 0,Y 666.314,Z 663.19,A -85,B 0,C 180,E1 4522.092,E2 4522.092} C_VEL
LIN {X 0,Y 666.669,Z 663.19,A -85,B 0,C 180,E1 4530.83,E2 4530.83} C_VEL
LIN {X 0,Y 666.357,Z 663.19,A -85,B 0,C 180,E1 4538.802,E2 4538.802} C_VEL
LIN {X 0,Y 666.04,Z 663.19,A -85,B 0,C 180,E1 4546.02,E2 4546.02} C_VEL
LIN {X 0,Y 666.599,Z 663.545,A -85,B 0,C 180,E1 4551.651,E2 4551.651} C_VEL
LIN {X 0,Y 684.06,Z 701.591,A -85,B 0,C 180,E1 4553.289,E2 4553.289} C_VEL
LIN {X 0,Y 682.45,Z 774.919,A -85,B 0,C 180,E1 4554.699,E2 4554.699} C_VEL
LIN {X 0,Y 678.979,Z 843.693,A -85,B 0,C 180,E1 4557.249,E2 4557.249} C_VEL
LIN {X 0,Y 674.705,Z 910.675,A -85,B 0,C 180,E1 4561.18,E2 4561.18} C_VEL
LIN {X 0,Y 670.96,Z 968.989,A -85,B 0,C 180,E1 4566.237,E2 4566.237} C_VEL
LIN {X 0,Y 668.547,Z 1013.602,A -85,B 0,C 180,E1 4571.828,E2 4571.828} C_VEL
LIN {X 0,Y 667.248,Z 1044.385,A -85,B 0,C 180,E1 4577.532,E2 4577.532} C_VEL
LIN {X 0,Y 666.858,Z 1061.848,A -85,B 0,C 180,E1 4582.816,E2 4582.816} C_VEL
LIN {X 0,Y 666.706,Z 1069.803,A -85,B 0,C 180,E1 4588.045,E2 4588.045} C_VEL
LIN {X 0,Y 666.862,Z 1068.733,A -85,B 0,C 180,E1 4593.259,E2 4593.259} C_VEL
LIN {X 0,Y 667.008,Z 1058.416,A -85,B 0,C 180,E1 4598.498,E2 4598.498} C_VEL
LIN {X 0,Y 667.571,Z 1035.771,A -85,B 0,C 180,E1 4604.335,E2 4604.335} C_VEL
LIN {X 0,Y 669.089,Z 1000.525,A -85,B 0,C 180,E1 4610.05,E2 4610.05} C_VEL
LIN {X 0,Y 672.152,Z 949.955,A -85,B 0,C 180,E1 4615.623,E2 4615.623} C_VEL
LIN {X 0,Y 676.157,Z 888.508,A -85,B 0,C 180,E1 4620.306,E2 4620.306} C_VEL
LIN {X 0,Y 680.293,Z 821.219,A -85,B 0,C 180,E1 4623.733,E2 4623.733} C_VEL
LIN {X 0,Y 683.345,Z 750.794,A -85,B 0,C 180,E1 4625.896,E2 4625.896} C_VEL
LIN {X 0,Y 682.684,Z 694.295,A -85,B 0,C 180,E1 4626.891,E2 4626.891} C_VEL
LIN {X 0,Y 666.302,Z 663.19,A -85,B 0,C 180,E1 4628.492,E2 4628.492} C_VEL
LIN {X 0,Y 666.325,Z 663.19,A -85,B 0,C 180,E1 4635.974,E2 4635.974} C_VEL
LIN {X 0,Y 666.313,Z 663.19,A -85,B 0,C 180,E1 4644.471,E2 4644.471} C_VEL
LIN {X 0,Y 666.529,Z 663.19,A -85,B 0,C 180,E1 4652.156,E2 4652.156} C_VEL
LIN {X 0,Y 666.654,Z 663.19,A -85,B 0,C 180,E1 4660.733,E2 4660.733} C_VEL
LIN {X 0,Y 666.818,Z 663.19,A -85,B 0,C 180,E1 4668.83,E2 4668.83} C_VEL
LIN {X 0,Y 666.832,Z 663.19,A -85,B 0,C 180,E1 4676.724,E2 4676.724} C_VEL
LIN {X 0,Y 666.661,Z 663.19,A -85,B 0,C 180,E1 4684.556,E2 4684.556} C_VEL
LIN {X 0,Y 666.489,Z 663.19,A -85,B 0,C 180,E1 4692.48,E2 4692.48} C_VEL
LIN {X 0,Y 666.513,Z 663.19,A -85,B 0,C 180,E1 4700.654,E2 4700.654} C_VEL
LIN {X 0,Y 666.4,Z 663.19,A -85,B 0,C 180,E1 4708.827,E2 4708.827} C_VEL
LIN {X 0,Y 666.515,Z 663.19,A -85,B 0,C 180,E1 4717.1,E2 4717.1} C_VEL
LIN {X 0,Y 666.4,Z 663.19,A -85,B 0,C 180,E1 4726.049,E2 4726.049} C_VEL
LIN {X 0,Y 666.983,Z 664.774,A -85,B 0,C 180,E1 4728.783,E2 4728.783} C_VEL
LIN {X 0,Y 683.973,Z 701.141,A -85,B 0,C 180,E1 4730.364,E2 4730.364} C_VEL
LIN {X 0,Y 681.96,Z 776.982,A -85,B 0,C 180,E1 4732.006,E2 4732.006} C_VEL
LIN {X 0,Y 678.293,Z 846.012,A -85,B 0,C 180,E1 4734.81,E2 4734.81} C_VEL
LIN {X 0,Y 674.101,Z 911.575,A -85,B 0,C 180,E1 4738.953,E2 4738.953} C_VEL
LIN {X 0,Y 670.62,Z 966.891,A -85,B 0,C 180,E1 4744.046,E2 4744.046} C_VEL
LIN {X 0,Y 668.504,Z 1010.91,A -85,B 0,C 180,E1 4749.938,E2 4749.938} C_VEL
LIN {X 0,Y 667.703,Z 1041.103,A -85,B 0,C 180,E1 4756.204,E2 4756.204} C_VEL
LIN {X 0,Y 667.302,Z 1057.582,A -85,B 0,C 180,E1 4762.82,E2 4762.82} C_VEL
LIN {X 0,Y 667.134,Z 1059.46,A -85,B 0,C 180,E1 4769.349,E2 4769.349} C_VEL
LIN {X 0,Y 666.888,Z 1057.453,A -85,B 0,C 180,E1 4771.153,E2 4771.153} C_VEL
LIN {X 0,Y 659.543,Z 1052.059,A -85,B 0,C 180,E1 4774.13,E2 4774.13} C_VEL
LIN {X 0,Y 659.772,Z 1029.818,A -85,B 0,C 180,E1 4780.595,E2 4780.595} C_VEL
LIN {X 0,Y 661.244,Z 994.696,A -85,B 0,C 180,E1 4786.658,E2 4786.658} C_VEL
LIN {X 0,Y 664.282,Z 946.062,A -85,B 0,C 180,E1 4792.314,E2 4792.314} C_VEL
LIN {X 0,Y 668.641,Z 885.602,A -85,B 0,C 180,E1 4797.156,E2 4797.156} C_VEL
LIN {X 0,Y 673.09,Z 818.1,A -85,B 0,C 180,E1 4800.786,E2 4800.786} C_VEL
LIN {X 0,Y 676.534,Z 745.571,A -85,B 0,C 180,E1 4803.15,E2 4803.15} C_VEL
LIN {X 0,Y 676.391,Z 698.911,A -85,B 0,C 180,E1 4804.057,E2 4804.057} C_VEL
LIN {X 0,Y 658.551,Z 663.19,A -85,B 0,C 180,E1 4805.784,E2 4805.784} C_VEL
LIN {X 0,Y 658.396,Z 663.19,A -85,B 0,C 180,E1 4815.343,E2 4815.343} C_VEL
LIN {X 0,Y 658.367,Z 663.19,A -85,B 0,C 180,E1 4824.012,E2 4824.012} C_VEL
LIN {X 0,Y 658.392,Z 663.19,A -85,B 0,C 180,E1 4832.465,E2 4832.465} C_VEL
LIN {X 0,Y 658.365,Z 663.19,A -85,B 0,C 180,E1 4840.486,E2 4840.486} C_VEL
LIN {X 0,Y 659.345,Z 663.19,A -85,B 0,C 180,E1 4848.731,E2 4848.731} C_VEL
LIN {X 0,Y 659.122,Z 663.19,A -85,B 0,C 180,E1 4858.035,E2 4858.035} C_VEL
LIN {X 0,Y 658.928,Z 663.19,A -85,B 0,C 180,E1 4865.964,E2 4865.964} C_VEL
LIN {X 0,Y 658.614,Z 663.19,A -85,B 0,C 180,E1 4874.018,E2 4874.018} C_VEL
LIN {X 0,Y 658.238,Z 663.19,A -85,B 0,C 180,E1 4882.378,E2 4882.378} C_VEL
LIN {X 0,Y 658.673,Z 663.19,A -85,B 0,C 180,E1 4891.246,E2 4891.246} C_VEL
LIN {X 0,Y 658.361,Z 663.19,A -85,B 0,C 180,E1 4899.502,E2 4899.502} C_VEL
LIN {X 0,Y 658.083,Z 663.19,A -85,B 0,C 180,E1 4907.175,E2 4907.175} C_VEL
LIN {X 0,Y 658.842,Z 665.137,A -85,B 0,C 180,E1 4911.137,E2 4911.137} C_VEL
LIN {X 0,Y 677.635,Z 704.073,A -85,B 0,C 180,E1 4912.915,E2 4912.915} C_VEL
LIN {X 0,Y 675.749,Z 777.803,A -85,B 0,C 180,E1 4914.383,E2 4914.383} C_VEL
LIN {X 0,Y 671.924,Z 847.282,A -85,B 0,C 180,E1 4917.044,E2 4917.044} C_VEL
LIN {X 0,Y 667.255,Z 913.714,A -85,B 0,C 180,E1 4921.054,E2 4921.054} C_VEL
LIN {X 0,Y 663.266,Z 970.682,A -85,B 0,C 180,E1 4926.132,E2 4926.132} C_VEL
LIN {X 0,Y 660.635,Z 1015.801,A -85,B 0,C 180,E1 4931.949,E2 4931.949} C_VEL
LIN {X 0,Y 659.383,Z 1047.283,A -85,B 0,C 180,E1 4938.104,E2 4938.104} C_VEL
LIN {X 0,Y 659.225,Z 1064.712,A -85,B 0,C 180,E1 4944.059,E2 4944.059} C_VEL
LIN {X 0,Y 659.626,Z 1070.338,A -85,B 0,C 180,E1 4950.659,E2 4950.659} C_VEL
LIN {X 0,Y 659.394,Z 1061.847,A -85,B 0,C 180,E1 4957.267,E2 4957.267} C_VEL
LIN {X 0,Y 659.673,Z 1039.879,A -85,B 0,C 180,E1 4963.629,E2 4963.629} C_VEL
LIN {X 0,Y 661.153,Z 1005.026,A -85,B 0,C 180,E1 4969.658,E2 4969.658} C_VEL
LIN {X 0,Y 664.293,Z 956.049,A -85,B 0,C 180,E1 4975.36,E2 4975.36} C_VEL
LIN {X 0,Y 668.57,Z 895.669,A -85,B 0,C 180,E1 4980.2,E2 4980.2} C_VEL
LIN {X 0,Y 673.101,Z 828.094,A -85,B 0,C 180,E1 4983.83,E2 4983.83} C_VEL
LIN {X 0,Y 676.573,Z 756.021,A -85,B 0,C 180,E1 4986.181,E2 4986.181} C_VEL
LIN {X 0,Y 676.468,Z 697.529,A -85,B 0,C 180,E1 4987.245,E2 4987.245} C_VEL
LIN {X 0,Y 658.168,Z 663.19,A -85,B 0,C 180,E1 4989.004,E2 4989.004} C_VEL
LIN {X 0,Y 658.003,Z 663.19,A -85,B 0,C 180,E1 4997.101,E2 4997.101} C_VEL
LIN {X 0,Y 658.122,Z 663.19,A -85,B 0,C 180,E1 5005.578,E2 5005.578} C_VEL
LIN {X 0,Y 658.282,Z 663.19,A -85,B 0,C 180,E1 5013.266,E2 5013.266} C_VEL
LIN {X 0,Y 658.34,Z 663.19,A -85,B 0,C 180,E1 5021.851,E2 5021.851} C_VEL
LIN {X 0,Y 658.472,Z 663.19,A -85,B 0,C 180,E1 5030.03,E2 5030.03} C_VEL
LIN {X 0,Y 658.855,Z 663.19,A -85,B 0,C 180,E1 5036.684,E2 5036.684} C_VEL
LIN {X 0,Y 658.652,Z 663.19,A -85,B 0,C 180,E1 5044.612,E2 5044.612} C_VEL
LIN {X 0,Y 658.451,Z 663.19,A -85,B 0,C 180,E1 5052.635,E2 5052.635} C_VEL
LIN {X 0,Y 658.446,Z 663.19,A -85,B 0,C 180,E1 5060.919,E2 5060.919} C_VEL
LIN {X 0,Y 658.463,Z 663.19,A -85,B 0,C 180,E1 5068.183,E2 5068.183} C_VEL
LIN {X 0,Y 658.472,Z 663.19,A -85,B 0,C 180,E1 5075.982,E2 5075.982} C_VEL
LIN {X 0,Y 658.05,Z 663.19,A -85,B 0,C 180,E1 5083.457,E2 5083.457} C_VEL
LIN {X 0,Y 658.97,Z 664.972,A -85,B 0,C 180,E1 5088.236,E2 5088.236} C_VEL
LIN {X 0,Y 677.529,Z 702.486,A -85,B 0,C 180,E1 5089.979,E2 5089.979} C_VEL
LIN {X 0,Y 675.252,Z 778.38,A -85,B 0,C 180,E1 5091.657,E2 5091.657} C_VEL
LIN {X 0,Y 671.184,Z 848.406,A -85,B 0,C 180,E1 5094.563,E2 5094.563} C_VEL
LIN {X 0,Y 666.6,Z 913.942,A -85,B 0,C 180,E1 5098.8,E2 5098.8} C_VEL
LIN {X 0,Y 662.871,Z 969.162,A -85,B 0,C 180,E1 5104.019,E2 5104.019} C_VEL
LIN {X 0,Y 660.598,Z 1013.181,A -85,B 0,C 180,E1 5110.123,E2 5110.123} C_VEL
LIN {X 0,Y 659.794,Z 1043.308,A -85,B 0,C 180,E1 5116.713,E2 5116.713} C_VEL
LIN {X 0,Y 659.31,Z 1057.533,A -85,B 0,C 180,E1 5122.732,E2 5122.732} C_VEL
LIN {X 0,Y 659.153,Z 1059.488,A -85,B 0,C 180,E1 5129.341,E2 5129.341} C_VEL
LIN {X 0,Y 659.543,Z 1052.059,A -85,B 0,C 180,E1 5134.13,E2 5134.13} C_VEL
LIN {X 0,Y 651.135,Z 1044.22,A -85,B 0,C 180,E1 5137.066,E2 5137.066} C_VEL
LIN {X 0,Y 651.934,Z 1020.079,A -85,B 0,C 180,E1 5142.766,E2 5142.766} C_VEL
LIN {X 0,Y 654.089,Z 982.26,A -85,B 0,C 180,E1 5148.588,E2 5148.588} C_VEL
LIN {X 0,Y 657.89,Z 929.952,A -85,B 0,C 180,E1 5154.124,E2 5154.124} C_VEL
LIN {X 0,Y 662.92,Z 866.615,A -85,B 0,C 180,E1 5158.708,E2 5158.708} C_VEL
LIN {X 0,Y 667.594,Z 798.066,A -85,B 0,C 180,E1 5161.975,E2 5161.975} C_VEL
LIN {X 0,Y 670.763,Z 730.117,A -85,B 0,C 180,E1 5163.875,E2 5163.875} C_VEL
LIN {X 0,Y 669.84,Z 701.47,A -85,B 0,C 180,E1 5164.444,E2 5164.444} C_VEL
LIN {X 0,Y 650.48,Z 663.19,A -85,B 0,C 180,E1 5166.474,E2 5166.474} C_VEL
LIN {X 0,Y 650.395,Z 663.19,A -85,B 0,C 180,E1 5175.325,E2 5175.325} C_VEL
LIN {X 0,Y 650.384,Z 663.19,A -85,B 0,C 180,E1 5183.551,E2 5183.551} C_VEL
LIN {X 0,Y 650.472,Z 663.19,A -85,B 0,C 180,E1 5191.44,E2 5191.44} C_VEL
LIN {X 0,Y 650.397,Z 663.19,A -85,B 0,C 180,E1 5200.237,E2 5200.237} C_VEL
LIN {X 0,Y 651.339,Z 663.19,A -85,B 0,C 180,E1 5208.591,E2 5208.591} C_VEL
LIN {X 0,Y 651.125,Z 663.19,A -85,B 0,C 180,E1 5218.011,E2 5218.011} C_VEL
LIN {X 0,Y 650.883,Z 663.19,A -85,B 0,C 180,E1 5226.038,E2 5226.038} C_VEL
LIN {X 0,Y 650.389,Z 663.19,A -85,B 0,C 180,E1 5234.628,E2 5234.628} C_VEL
LIN {X 0,Y 650.12,Z 663.19,A -85,B 0,C 180,E1 5242.878,E2 5242.878} C_VEL
LIN {X 0,Y 650.65,Z 663.19,A -85,B 0,C 180,E1 5251.716,E2 5251.716} C_VEL
LIN {X 0,Y 650.346,Z 663.19,A -85,B 0,C 180,E1 5259.945,E2 5259.945} C_VEL
LIN {X 0,Y 650.213,Z 663.19,A -85,B 0,C 180,E1 5268.343,E2 5268.343} C_VEL
LIN {X 0,Y 650.684,Z 664.87,A -85,B 0,C 180,E1 5270.554,E2 5270.554} C_VEL
LIN {X 0,Y 671.255,Z 706.939,A -85,B 0,C 180,E1 5272.54,E2 5272.54} C_VEL
LIN {X 0,Y 669.094,Z 779.815,A -85,B 0,C 180,E1 5274.035,E2 5274.035} C_VEL
LIN {X 0,Y 664.916,Z 849.769,A -85,B 0,C 180,E1 5276.78,E2 5276.78} C_VEL
LIN {X 0,Y 659.874,Z 915.381,A -85,B 0,C 180,E1 5280.834,E2 5280.834} C_VEL
LIN {X 0,Y 655.496,Z 973.238,A -85,B 0,C 180,E1 5286.119,E2 5286.119} C_VEL
LIN {X 0,Y 652.748,Z 1017.58,A -85,B 0,C 180,E1 5292.01,E2 5292.01} C_VEL
LIN {X 0,Y 651.475,Z 1048.523,A -85,B 0,C 180,E1 5298.274,E2 5298.274} C_VEL
LIN {X 0,Y 651.484,Z 1065.921,A -85,B 0,C 180,E1 5304.658,E2 5304.658} C_VEL
LIN {X 0,Y 651.619,Z 1070.338,A -85,B 0,C 180,E1 5310.667,E2 5310.667} C_VEL
LIN {X 0,Y 651.356,Z 1061.847,A -85,B 0,C 180,E1 5317.357,E2 5317.357} C_VEL
LIN {X 0,Y 651.704,Z 1039.88,A -85,B 0,C 180,E1 5323.798,E2 5323.798} C_VEL
LIN {X 0,Y 653.312,Z 1006.056,A -85,B 0,C 180,E1 5329.754,E2 5329.754} C_VEL
LIN {X 0,Y 656.651,Z 957.9,A -85,B 0,C 180,E1 5335.484,E2 5335.484} C_VEL
LIN {X 0,Y 661.308,Z 897.702,A -85,B 0,C 180,E1 5340.427,E2 5340.427} C_VEL
LIN {X 0,Y 666.178,Z 830.856,A -85,B 0,C 180,E1 5344.103,E2 5344.103} C_VEL
LIN {X 0,Y 669.92,Z 759.744,A -85,B 0,C 180,E1 5346.503,E2 5346.503} C_VEL
LIN {X 0,Y 669.916,Z 700.161,A -85,B 0,C 180,E1 5347.638,E2 5347.638} C_VEL
LIN {X 0,Y 650.047,Z 663.19,A -85,B 0,C 180,E1 5349.606,E2 5349.606} C_VEL
LIN {X 0,Y 649.976,Z 663.19,A -85,B 0,C 180,E1 5357.3,E2 5357.3} C_VEL
LIN {X 0,Y 650.057,Z 663.19,A -85,B 0,C 180,E1 5365.907,E2 5365.907} C_VEL
LIN {X 0,Y 650.101,Z 663.19,A -85,B 0,C 180,E1 5373.903,E2 5373.903} C_VEL
LIN {X 0,Y 650.362,Z 663.19,A -85,B 0,C 180,E1 5381.62,E2 5381.62} C_VEL
LIN {X 0,Y 650.489,Z 663.19,A -85,B 0,C 180,E1 5389.907,E2 5389.907} C_VEL
LIN {X 0,Y 650.864,Z 663.19,A -85,B 0,C 180,E1 5396.643,E2 5396.643} C_VEL
LIN {X 0,Y 650.623,Z 663.19,A -85,B 0,C 180,E1 5404.669,E2 5404.669} C_VEL
LIN {X 0,Y 650.398,Z 663.19,A -85,B 0,C 180,E1 5412.794,E2 5412.794} C_VEL
LIN {X 0,Y 650.668,Z 663.19,A -85,B 0,C 180,E1 5419.754,E2 5419.754} C_VEL
LIN {X 0,Y 650.393,Z 663.19,A -85,B 0,C 180,E1 5428.564,E2 5428.564} C_VEL
LIN {X 0,Y 650.456,Z 663.19,A -85,B 0,C 180,E1 5436.496,E2 5436.496} C_VEL
LIN {X 0,Y 650.244,Z 663.19,A -85,B 0,C 180,E1 5445.371,E2 5445.371} C_VEL
LIN {X 0,Y 650.801,Z 664.444,A -85,B 0,C 180,E1 5447.649,E2 5447.649} C_VEL
LIN {X 0,Y 671.028,Z 707.376,A -85,B 0,C 180,E1 5449.636,E2 5449.636} C_VEL
LIN {X 0,Y 668.396,Z 782.82,A -85,B 0,C 180,E1 5451.398,E2 5451.398} C_VEL
LIN {X 0,Y 663.905,Z 853.36,A -85,B 0,C 180,E1 5454.446,E2 5454.446} C_VEL
LIN {X 0,Y 659.094,Z 916.96,A -85,B 0,C 180,E1 5458.697,E2 5458.697} C_VEL
LIN {X 0,Y 655.054,Z 971.693,A -85,B 0,C 180,E1 5464.038,E2 5464.038} C_VEL
LIN {X 0,Y 652.742,Z 1015.441,A -85,B 0,C 180,E1 5470.314,E2 5470.314} C_VEL
LIN {X 0,Y 651.788,Z 1044.337,A -85,B 0,C 180,E1 5476.889,E2 5476.889} C_VEL
LIN {X 0,Y 651.321,Z 1057.484,A -85,B 0,C 180,E1 5482.643,E2 5482.643} C_VEL
LIN {X 0,Y 651.153,Z 1059.517,A -85,B 0,C 180,E1 5489.333,E2 5489.333} C_VEL
LIN {X 0,Y 651.142,Z 1049.322,A -85,B 0,C 180,E1 5495.345,E2 5495.345} C_VEL
LIN {X 0,Y 651.135,Z 1044.22,A -85,B 0,C 180,E1 5497.066,E2 5497.066} C_VEL
LIN {X 0,Y 644.004,Z 1033.824,A -85,B 0,C 180,E1 5500.018,E2 5500.018} C_VEL
LIN {X 0,Y 645.525,Z 998.808,A -85,B 0,C 180,E1 5506.548,E2 5506.548} C_VEL
LIN {X 0,Y 649,Z 949.86,A -85,B 0,C 180,E1 5512.555,E2 5512.555} C_VEL
LIN {X 0,Y 654.063,Z 890.302,A -85,B 0,C 180,E1 5517.563,E2 5517.563} C_VEL
LIN {X 0,Y 659.298,Z 823.031,A -85,B 0,C 180,E1 5521.362,E2 5521.362} C_VEL
LIN {X 0,Y 663.28,Z 751.084,A -85,B 0,C 180,E1 5523.849,E2 5523.849} C_VEL
LIN {X 0,Y 663.247,Z 704.06,A -85,B 0,C 180,E1 5524.841,E2 5524.841} C_VEL
LIN {X 0,Y 642.329,Z 663.19,A -85,B 0,C 180,E1 5527.013,E2 5527.013} C_VEL
LIN {X 0,Y 642.339,Z 663.19,A -85,B 0,C 180,E1 5536.057,E2 5536.057} C_VEL
LIN {X 0,Y 642.188,Z 663.19,A -85,B 0,C 180,E1 5544.634,E2 5544.634} C_VEL
LIN {X 0,Y 642.315,Z 663.19,A -85,B 0,C 180,E1 5552.579,E2 5552.579} C_VEL
LIN {X 0,Y 642.407,Z 663.19,A -85,B 0,C 180,E1 5559.981,E2 5559.981} C_VEL
LIN {X 0,Y 643.321,Z 663.19,A -85,B 0,C 180,E1 5568.446,E2 5568.446} C_VEL
LIN {X 0,Y 643.147,Z 663.19,A -85,B 0,C 180,E1 5577.986,E2 5577.986} C_VEL
LIN {X 0,Y 642.859,Z 663.19,A -85,B 0,C 180,E1 5586.114,E2 5586.114} C_VEL
LIN {X 0,Y 642.495,Z 663.19,A -85,B 0,C 180,E1 5594.377,E2 5594.377} C_VEL
LIN {X 0,Y 642.096,Z 663.19,A -85,B 0,C 180,E1 5602.972,E2 5602.972} C_VEL
LIN {X 0,Y 642.65,Z 663.19,A -85,B 0,C 180,E1 5610.542,E2 5610.542} C_VEL
LIN {X 0,Y 642.316,Z 663.19,A -85,B 0,C 180,E1 5618.789,E2 5618.789} C_VEL
LIN {X 0,Y 642.029,Z 663.19,A -85,B 0,C 180,E1 5626.161,E2 5626.161} C_VEL
LIN {X 0,Y 642.503,Z 664.516,A -85,B 0,C 180,E1 5629.948,E2 5629.948} C_VEL
LIN {X 0,Y 664.871,Z 710.786,A -85,B 0,C 180,E1 5632.171,E2 5632.171} C_VEL
LIN {X 0,Y 662.422,Z 783.165,A -85,B 0,C 180,E1 5633.724,E2 5633.724} C_VEL
LIN {X 0,Y 657.907,Z 851.968,A -85,B 0,C 180,E1 5636.499,E2 5636.499} C_VEL
LIN {X 0,Y 652.464,Z 917.426,A -85,B 0,C 180,E1 5640.64,E2 5640.64} C_VEL
LIN {X 0,Y 647.771,Z 975.029,A -85,B 0,C 180,E1 5646.022,E2 5646.022} C_VEL
LIN {X 0,Y 644.845,Z 1019.129,A -85,B 0,C 180,E1 5652.034,E2 5652.034} C_VEL
LIN {X 0,Y 643.54,Z 1049.762,A -85,B 0,C 180,E1 5658.446,E2 5658.446} C_VEL
LIN {X 0,Y 643.565,Z 1067.018,A -85,B 0,C 180,E1 5665.27,E2 5665.27} C_VEL
LIN {X 0,Y 643.244,Z 1069.804,A -85,B 0,C 180,E1 5672.027,E2 5672.027} C_VEL
LIN {X 0,Y 643.075,Z 1059.742,A -85,B 0,C 180,E1 5678.347,E2 5678.347} C_VEL
LIN {X 0,Y 643.741,Z 1038.331,A -85,B 0,C 180,E1 5684.321,E2 5684.321} C_VEL
LIN {X 0,Y 645.541,Z 1004.221,A -85,B 0,C 180,E1 5690.273,E2 5690.273} C_VEL
LIN {X 0,Y 649.295,Z 955.959,A -85,B 0,C 180,E1 5695.998,E2 5695.998} C_VEL
LIN {X 0,Y 654.35,Z 895.089,A -85,B 0,C 180,E1 5700.969,E2 5700.969} C_VEL
LIN {X 0,Y 659.637,Z 827.721,A -85,B 0,C 180,E1 5704.635,E2 5704.635} C_VEL
LIN {X 0,Y 663.68,Z 755.795,A -85,B 0,C 180,E1 5707.005,E2 5707.005} C_VEL
LIN {X 0,Y 663.643,Z 703.249,A -85,B 0,C 180,E1 5708.015,E2 5708.015} C_VEL
LIN {X 0,Y 641.979,Z 663.19,A -85,B 0,C 180,E1 5710.168,E2 5710.168} C_VEL
LIN {X 0,Y 641.86,Z 663.19,A -85,B 0,C 180,E1 5718.091,E2 5718.091} C_VEL
LIN {X 0,Y 642.016,Z 663.19,A -85,B 0,C 180,E1 5726.233,E2 5726.233} C_VEL
LIN {X 0,Y 642.07,Z 663.19,A -85,B 0,C 180,E1 5734.051,E2 5734.051} C_VEL
LIN {X 0,Y 642.407,Z 663.19,A -85,B 0,C 180,E1 5741.385,E2 5741.385} C_VEL
LIN {X 0,Y 642.508,Z 663.19,A -85,B 0,C 180,E1 5749.78,E2 5749.78} C_VEL
LIN {X 0,Y 642.887,Z 663.19,A -85,B 0,C 180,E1 5756.602,E2 5756.602} C_VEL
LIN {X 0,Y 642.596,Z 663.19,A -85,B 0,C 180,E1 5764.727,E2 5764.727} C_VEL
LIN {X 0,Y 642.378,Z 663.19,A -85,B 0,C 180,E1 5772.956,E2 5772.956} C_VEL
LIN {X 0,Y 642.408,Z 663.19,A -85,B 0,C 180,E1 5781.187,E2 5781.187} C_VEL
LIN {X 0,Y 642.367,Z 663.19,A -85,B 0,C 180,E1 5788.955,E2 5788.955} C_VEL
LIN {X 0,Y 642.406,Z 663.19,A -85,B 0,C 180,E1 5797.029,E2 5797.029} C_VEL
LIN {X 0,Y 642.371,Z 663.19,A -85,B 0,C 180,E1 5806.087,E2 5806.087} C_VEL
LIN {X 0,Y 642.835,Z 665.367,A -85,B 0,C 180,E1 5807.077,E2 5807.077} C_VEL
LIN {X 0,Y 664.674,Z 707.917,A -85,B 0,C 180,E1 5809.226,E2 5809.226} C_VEL
LIN {X 0,Y 661.809,Z 783.05,A -85,B 0,C 180,E1 5810.998,E2 5810.998} C_VEL
LIN {X 0,Y 657.013,Z 853.118,A -85,B 0,C 180,E1 5814.048,E2 5814.048} C_VEL
LIN {X 0,Y 651.72,Z 917.946,A -85,B 0,C 180,E1 5818.431,E2 5818.431} C_VEL
LIN {X 0,Y 647.291,Z 973.278,A -85,B 0,C 180,E1 5823.943,E2 5823.943} C_VEL
LIN {X 0,Y 644.829,Z 1016.257,A -85,B 0,C 180,E1 5830.251,E2 5830.251} C_VEL
LIN {X 0,Y 643.737,Z 1045.358,A -85,B 0,C 180,E1 5837.068,E2 5837.068} C_VEL
LIN {X 0,Y 642.929,Z 1059.03,A -85,B 0,C 180,E1 5843.907,E2 5843.907} C_VEL
LIN {X 0,Y 643.154,Z 1059.546,A -85,B 0,C 180,E1 5849.324,E2 5849.324} C_VEL
LIN {X 0,Y 643.132,Z 1049.431,A -85,B 0,C 180,E1 5855.412,E2 5855.412} C_VEL
LIN {X 0,Y 644.004,Z 1033.824,A -85,B 0,C 180,E1 5860.018,E2 5860.018} C_VEL
LIN {X 0,Y 636.086,Z 1021.376,A -85,B 0,C 180,E1 5862.909,E2 5862.909} C_VEL
LIN {X 0,Y 638.554,Z 984.199,A -85,B 0,C 180,E1 5868.878,E2 5868.878} C_VEL
LIN {X 0,Y 642.893,Z 932.78,A -85,B 0,C 180,E1 5874.544,E2 5874.544} C_VEL
LIN {X 0,Y 648.718,Z 869.485,A -85,B 0,C 180,E1 5879.302,E2 5879.302} C_VEL
LIN {X 0,Y 654.137,Z 801.248,A -85,B 0,C 180,E1 5882.671,E2 5882.671} C_VEL
LIN {X 0,Y 657.915,Z 732.43,A -85,B 0,C 180,E1 5884.671,E2 5884.671} C_VEL
LIN {X 0,Y 656.999,Z 707.089,A -85,B 0,C 180,E1 5885.217,E2 5885.217} C_VEL
LIN {X 0,Y 634.242,Z 663.19,A -85,B 0,C 180,E1 5887.566,E2 5887.566} C_VEL
LIN {X 0,Y 634.169,Z 663.19,A -85,B 0,C 180,E1 5897.012,E2 5897.012} C_VEL
LIN {X 0,Y 634.074,Z 663.19,A -85,B 0,C 180,E1 5905.788,E2 5905.788} C_VEL
LIN {X 0,Y 634.274,Z 663.19,A -85,B 0,C 180,E1 5913.741,E2 5913.741} C_VEL
LIN {X 0,Y 634.284,Z 663.19,A -85,B 0,C 180,E1 5921.169,E2 5921.169} C_VEL
LIN {X 0,Y 635.334,Z 663.19,A -85,B 0,C 180,E1 5928.299,E2 5928.299} C_VEL
LIN {X 0,Y 635.148,Z 663.19,A -85,B 0,C 180,E1 5937.961,E2 5937.961} C_VEL
LIN {X 0,Y 634.817,Z 663.19,A -85,B 0,C 180,E1 5946.191,E2 5946.191} C_VEL
LIN {X 0,Y 634.436,Z 663.19,A -85,B 0,C 180,E1 5954.564,E2 5954.564} C_VEL
LIN {X 0,Y 634.112,Z 663.19,A -85,B 0,C 180,E1 5962.974,E2 5962.974} C_VEL
LIN {X 0,Y 634.627,Z 663.19,A -85,B 0,C 180,E1 5970.961,E2 5970.961} C_VEL
LIN {X 0,Y 634.318,Z 663.19,A -85,B 0,C 180,E1 5979.372,E2 5979.372} C_VEL
LIN {X 0,Y 634.033,Z 663.19,A -85,B 0,C 180,E1 5987.029,E2 5987.029} C_VEL
LIN {X 0,Y 634.565,Z 665.212,A -85,B 0,C 180,E1 5989.355,E2 5989.355} C_VEL
LIN {X 0,Y 658.516,Z 712.464,A -85,B 0,C 180,E1 5991.768,E2 5991.768} C_VEL
LIN {X 0,Y 655.817,Z 784.755,A -85,B 0,C 180,E1 5993.358,E2 5993.358} C_VEL
LIN {X 0,Y 650.974,Z 853.067,A -85,B 0,C 180,E1 5996.159,E2 5996.159} C_VEL
LIN {X 0,Y 645.214,Z 918.066,A -85,B 0,C 180,E1 6000.331,E2 6000.331} C_VEL
LIN {X 0,Y 640.113,Z 975.758,A -85,B 0,C 180,E1 6005.801,E2 6005.801} C_VEL
LIN {X 0,Y 636.984,Z 1018.792,A -85,B 0,C 180,E1 6011.749,E2 6011.749} C_VEL
LIN {X 0,Y 635.538,Z 1049.761,A -85,B 0,C 180,E1 6018.299,E2 6018.299} C_VEL
LIN {X 0,Y 635.553,Z 1067.018,A -85,B 0,C 180,E1 6025.21,E2 6025.21} C_VEL
LIN {X 0,Y 635.23,Z 1069.804,A -85,B 0,C 180,E1 6032.052,E2 6032.052} C_VEL
LIN {X 0,Y 635.108,Z 1060.28,A -85,B 0,C 180,E1 6038.237,E2 6038.237} C_VEL
LIN {X 0,Y 635.776,Z 1039.881,A -85,B 0,C 180,E1 6044.151,E2 6044.151} C_VEL
LIN {X 0,Y 637.624,Z 1006.637,A -85,B 0,C 180,E1 6050.173,E2 6050.173} C_VEL
LIN {X 0,Y 641.637,Z 958.1,A -85,B 0,C 180,E1 6056.103,E2 6056.103} C_VEL
LIN {X 0,Y 646.92,Z 899.285,A -85,B 0,C 180,E1 6061.062,E2 6061.062} C_VEL
LIN {X 0,Y 652.671,Z 831.74,A -85,B 0,C 180,E1 6064.868,E2 6064.868} C_VEL
LIN {X 0,Y 657.087,Z 759.624,A -85,B 0,C 180,E1 6067.339,E2 6067.339} C_VEL
LIN {X 0,Y 657.152,Z 706.073,A -85,B 0,C 180,E1 6068.42,E2 6068.42} C_VEL
LIN {X 0,Y 633.953,Z 663.19,A -85,B 0,C 180,E1 6070.885,E2 6070.885} C_VEL
LIN {X 0,Y 633.766,Z 663.19,A -85,B 0,C 180,E1 6078.912,E2 6078.912} C_VEL
LIN {X 0,Y 634.012,Z 663.19,A -85,B 0,C 180,E1 6085.748,E2 6085.748} C_VEL
LIN {X 0,Y 634.105,Z 663.19,A -85,B 0,C 180,E1 6093.739,E2 6093.739} C_VEL
LIN {X 0,Y 634.404,Z 663.19,A -85,B 0,C 180,E1 6101.141,E2 6101.141} C_VEL
LIN {X 0,Y 634.533,Z 663.19,A -85,B 0,C 180,E1 6109.65,E2 6109.65} C_VEL
LIN {X 0,Y 634.894,Z 663.19,A -85,B 0,C 180,E1 6116.559,E2 6116.559} C_VEL
LIN {X 0,Y 634.569,Z 663.19,A -85,B 0,C 180,E1 6124.787,E2 6124.787} C_VEL
LIN {X 0,Y 634.334,Z 663.19,A -85,B 0,C 180,E1 6133.123,E2 6133.123} C_VEL
LIN {X 0,Y 634.522,Z 663.19,A -85,B 0,C 180,E1 6140.278,E2 6140.278} C_VEL
LIN {X 0,Y 634.443,Z 663.19,A -85,B 0,C 180,E1 6147.791,E2 6147.791} C_VEL
LIN {X 0,Y 634.382,Z 663.19,A -85,B 0,C 180,E1 6155.868,E2 6155.868} C_VEL
LIN {X 0,Y 634.043,Z 663.19,A -85,B 0,C 180,E1 6163.159,E2 6163.159} C_VEL
LIN {X 0,Y 634.616,Z 664.845,A -85,B 0,C 180,E1 6166.446,E2 6166.446} C_VEL
LIN {X 0,Y 658.242,Z 711.172,A -85,B 0,C 180,E1 6168.844,E2 6168.844} C_VEL
LIN {X 0,Y 655.017,Z 787.168,A -85,B 0,C 180,E1 6170.717,E2 6170.717} C_VEL
LIN {X 0,Y 649.721,Z 858.117,A -85,B 0,C 180,E1 6173.93,E2 6173.93} C_VEL
LIN {X 0,Y 644.072,Z 921.767,A -85,B 0,C 180,E1 6178.409,E2 6178.409} C_VEL
LIN {X 0,Y 639.471,Z 975.912,A -85,B 0,C 180,E1 6183.979,E2 6183.979} C_VEL
LIN {X 0,Y 636.914,Z 1017.292,A -85,B 0,C 180,E1 6190.227,E2 6190.227} C_VEL
LIN {X 0,Y 635.779,Z 1045.233,A -85,B 0,C 180,E1 6196.903,E2 6196.903} C_VEL
LIN {X 0,Y 634.943,Z 1059.001,A -85,B 0,C 180,E1 6203.83,E2 6203.83} C_VEL
LIN {X 0,Y 635.154,Z 1059.574,A -85,B 0,C 180,E1 6209.316,E2 6209.316} C_VEL
LIN {X 0,Y 635.124,Z 1049.539,A -85,B 0,C 180,E1 6215.48,E2 6215.48} C_VEL
LIN {X 0,Y 635.829,Z 1027.287,A -85,B 0,C 180,E1 6221.696,E2 6221.696} C_VEL
LIN {X 0,Y 636.086,Z 1021.376,A -85,B 0,C 180,E1 6222.909,E2 6222.909} C_VEL
LIN {X 0,Y 629.7,Z 1006.621,A -85,B 0,C 180,E1 6225.788,E2 6225.788} C_VEL
LIN {X 0,Y 633.252,Z 960.564,A -85,B 0,C 180,E1 6232.045,E2 6232.045} C_VEL
LIN {X 0,Y 638.668,Z 903.391,A -85,B 0,C 180,E1 6237.356,E2 6237.356} C_VEL
LIN {X 0,Y 644.489,Z 837.996,A -85,B 0,C 180,E1 6241.469,E2 6241.469} C_VEL
LIN {X 0,Y 649.62,Z 765.512,A -85,B 0,C 180,E1 6244.314,E2 6244.314} C_VEL
LIN {X 0,Y 650.605,Z 710.049,A -85,B 0,C 180,E1 6245.614,E2 6245.614} C_VEL
LIN {X 0,Y 626.089,Z 663.19,A -85,B 0,C 180,E1 6248.309,E2 6248.309} C_VEL
LIN {X 0,Y 626.167,Z 663.19,A -85,B 0,C 180,E1 6256.326,E2 6256.326} C_VEL
LIN {X 0,Y 626.093,Z 663.19,A -85,B 0,C 180,E1 6265.29,E2 6265.29} C_VEL
LIN {X 0,Y 626.268,Z 663.19,A -85,B 0,C 180,E1 6273.379,E2 6273.379} C_VEL
LIN {X 0,Y 626.337,Z 663.19,A -85,B 0,C 180,E1 6280.921,E2 6280.921} C_VEL
LIN {X 0,Y 627.34,Z 663.19,A -85,B 0,C 180,E1 6288.227,E2 6288.227} C_VEL
LIN {X 0,Y 627.166,Z 663.19,A -85,B 0,C 180,E1 6297.935,E2 6297.935} C_VEL
LIN {X 0,Y 626.786,Z 663.19,A -85,B 0,C 180,E1 6306.271,E2 6306.271} C_VEL
LIN {X 0,Y 626.37,Z 663.19,A -85,B 0,C 180,E1 6314.755,E2 6314.755} C_VEL
LIN {X 0,Y 626.257,Z 663.19,A -85,B 0,C 180,E1 6322.081,E2 6322.081} C_VEL
LIN {X 0,Y 626.608,Z 663.19,A -85,B 0,C 180,E1 6331.402,E2 6331.402} C_VEL
LIN {X 0,Y 626.286,Z 663.19,A -85,B 0,C 180,E1 6340.298,E2 6340.298} C_VEL
LIN {X 0,Y 626.326,Z 664.586,A -85,B 0,C 180,E1 6348.697,E2 6348.697} C_VEL
LIN {X 0,Y 652.172,Z 714.585,A -85,B 0,C 180,E1 6351.363,E2 6351.363} C_VEL
LIN {X 0,Y 649.139,Z 787.293,A -85,B 0,C 180,E1 6353.013,E2 6353.013} C_VEL
LIN {X 0,Y 643.933,Z 855.712,A -85,B 0,C 180,E1 6355.896,E2 6355.896} C_VEL
LIN {X 0,Y 637.891,Z 919.442,A -85,B 0,C 180,E1 6360.073,E2 6360.073} C_VEL
LIN {X 0,Y 632.544,Z 975.754,A -85,B 0,C 180,E1 6365.493,E2 6365.493} C_VEL
LIN {X 0,Y 629.083,Z 1020.141,A -85,B 0,C 180,E1 6371.739,E2 6371.739} C_VEL
LIN {X 0,Y 627.609,Z 1050.719,A -85,B 0,C 180,E1 6378.435,E2 6378.435} C_VEL
LIN {X 0,Y 627.562,Z 1067.018,A -85,B 0,C 180,E1 6385.149,E2 6385.149} C_VEL
LIN {X 0,Y 627.245,Z 1069.804,A -85,B 0,C 180,E1 6392.079,E2 6392.079} C_VEL
LIN {X 0,Y 627.112,Z 1060.28,A -85,B 0,C 180,E1 6398.343,E2 6398.343} C_VEL
LIN {X 0,Y 627.823,Z 1039.88,A -85,B 0,C 180,E1 6404.334,E2 6404.334} C_VEL
LIN {X 0,Y 629.882,Z 1006.635,A -85,B 0,C 180,E1 6410.431,E2 6410.431} C_VEL
LIN {X 0,Y 634.173,Z 957.989,A -85,B 0,C 180,E1 6416.446,E2 6416.446} C_VEL
LIN {X 0,Y 639.981,Z 897.991,A -85,B 0,C 180,E1 6421.534,E2 6421.534} C_VEL
LIN {X 0,Y 646.001,Z 831.698,A -85,B 0,C 180,E1 6425.283,E2 6425.283} C_VEL
LIN {X 0,Y 650.708,Z 759.842,A -85,B 0,C 180,E1 6427.763,E2 6427.763} C_VEL
LIN {X 0,Y 650.871,Z 709.128,A -85,B 0,C 180,E1 6428.816,E2 6428.816} C_VEL
LIN {X 0,Y 625.943,Z 663.19,A -85,B 0,C 180,E1 6431.443,E2 6431.443} C_VEL
LIN {X 0,Y 625.777,Z 663.19,A -85,B 0,C 180,E1 6439.984,E2 6439.984} C_VEL
LIN {X 0,Y 626.057,Z 663.19,A -85,B 0,C 180,E1 6448.567,E2 6448.567} C_VEL
